C07237=1053.526,42.373,-75.968,170.999,31.827,155.969
C07238=1053.520,42.124,-75.951,170.997,31.825,155.968
C07239=1053.514,41.874,-75.935,170.995,31.822,155.968
C07240=1053.507,41.624,-75.918,170.994,31.820,155.968
C07241=1053.501,41.376,-75.902,170.993,31.818,155.967
C07242=1053.495,41.126,-75.885,170.991,31.816,155.967
C07243=1053.489,40.877,-75.869,170.989,31.814,155.967
C07244=1053.482,40.628,-75.852,170.988,31.811,155.966
C07245=1053.476,40.378,-75.835,170.986,31.809,155.966
C07246=1053.470,40.129,-75.819,170.984,31.807,155.966
C07247=1053.464,39.880,-75.803,170.983,31.805,155.965
C07248=1053.459,39.630,-75.787,170.981,31.802,155.965
C07249=1053.452,39.381,-75.769,170.979,31.800,155.965
C07250=1053.446,39.131,-75.753,170.978,31.798,155.964
C07251=1053.440,38.882,-75.736,170.977,31.796,155.964
C07252=1053.435,38.632,-75.720,170.975,31.794,155.964
C07253=1053.428,38.382,-75.703,170.974,31.792,155.963
C07254=1053.422,38.134,-75.686,170.972,31.790,155.963
C07255=1053.416,37.884,-75.670,170.970,31.787,155.963
C07256=1053.410,37.635,-75.654,170.969,31.785,155.962
C07257=1053.403,37.386,-75.638,170.967,31.783,155.962
C07258=1053.397,37.136,-75.622,170.965,31.781,155.962
C07259=1053.391,36.886,-75.605,170.963,31.779,155.961
C07260=1053.385,36.637,-75.589,170.962,31.777,155.961
C07261=1053.378,36.388,-75.572,170.961,31.775,155.961
C07262=1053.372,36.139,-75.556,170.959,31.772,155.960
C07263=1053.366,35.889,-75.539,170.958,31.770,155.960
C07264=1053.359,35.640,-75.524,170.956,31.768,155.960
C07265=1053.353,35.391,-75.507,170.954,31.766,155.960
C07266=1053.347,35.141,-75.491,170.953,31.764,155.959
C07267=1053.341,34.892,-75.475,170.951,31.762,155.959
C07268=1053.335,34.642,-75.458,170.949,31.759,155.958
C07269=1053.328,34.393,-75.442,170.947,31.757,155.958
C07270=1053.322,34.143,-75.426,170.946,31.755,155.958
C07271=1053.316,33.894,-75.410,170.945,31.753,155.958
C07272=1053.310,33.645,-75.394,170.943,31.751,155.957
C07273=1053.304,33.395,-75.377,170.942,31.749,155.957
C07274=1053.298,33.145,-75.361,170.940,31.746,155.957
C07275=1053.291,32.896,-75.345,170.938,31.744,155.956
C07276=1053.285,32.647,-75.329,170.937,31.742,155.956
C07277=1053.279,32.398,-75.313,170.935,31.740,155.956
C07278=1053.273,32.148,-75.296,170.933,31.738,155.955
C07279=1053.267,31.899,-75.280,170.931,31.736,155.955
C07280=1053.261,31.650,-75.264,170.930,31.733,155.955
C07281=1053.254,31.400,-75.248,170.929,31.731,155.954
C07282=1053.248,31.151,-75.232,170.927,31.729,155.954
C07283=1053.242,30.901,-75.215,170.926,31.727,155.954
C07284=1053.236,30.652,-75.199,170.924,31.725,155.953
C07285=1053.230,30.403,-75.183,170.922,31.723,155.953
C07286=1053.224,30.153,-75.167,170.920,31.720,155.953
C07287=1053.217,29.868,-75.149,170.919,31.718,155.952
C07288=1053.209,29.582,-75.130,170.917,31.716,155.952
C07289=1053.203,29.296,-75.112,170.915,31.714,155.952
C07290=1053.196,29.011,-75.094,170.914,31.711,155.951
C07291=1053.189,28.761,-75.077,170.912,31.709,155.951
C07292=1053.184,28.511,-75.062,170.910,31.707,155.951
C07293=1053.177,28.262,-75.046,170.909,31.704,155.950
C07294=1053.171,28.012,-75.030,170.907,31.702,155.950
C07295=1053.165,27.763,-75.013,170.905,31.700,155.950
C07296=1053.158,27.514,-74.998,170.903,31.698,155.949
C07297=1053.153,27.264,-74.982,170.902,31.696,155.949
C07298=1053.146,27.015,-74.966,170.900,31.694,155.949
C07299=1053.140,26.765,-74.950,170.899,31.692,155.949
C07300=1053.134,26.516,-74.934,170.897,31.690,155.948
C07301=1053.127,26.267,-74.918,170.896,31.688,155.948
C07302=1053.122,26.017,-74.903,170.894,31.686,155.948
C07303=1053.114,25.767,-74.887,170.892,31.684,155.947
C07304=1053.108,25.518,-74.870,170.891,31.682,155.947
C07305=1053.103,25.269,-74.854,170.889,31.679,155.947
C07306=1053.096,25.019,-74.839,170.887,31.677,155.946
C07307=1053.090,24.770,-74.823,170.885,31.675,155.946
C07308=1053.084,24.521,-74.807,170.884,31.673,155.946
C07309=1053.078,24.271,-74.792,170.883,31.671,155.945
C07310=1053.071,24.022,-74.776,170.881,31.669,155.945
C07311=1053.065,23.772,-74.760,170.880,31.667,155.945
C07312=1053.059,23.523,-74.744,170.878,31.665,155.945
C07313=1053.053,23.273,-74.729,170.876,31.663,155.944
C07314=1053.047,23.024,-74.712,170.874,31.660,155.944
C07315=1053.040,22.775,-74.697,170.873,31.659,155.944
C07316=1053.035,22.525,-74.681,170.871,31.656,155.943
C07317=1053.028,22.276,-74.666,170.869,31.654,155.943
C07318=1053.022,22.026,-74.650,170.868,31.652,155.943
C07319=1053.016,21.777,-74.634,170.867,31.650,155.942
C07320=1053.010,21.528,-74.618,170.865,31.648,155.942
C07321=1053.003,21.278,-74.603,170.863,31.645,155.942
C07322=1052.997,21.029,-74.587,170.862,31.644,155.942
C07323=1052.991,20.779,-74.571,170.860,31.641,155.941
C07324=1052.985,20.530,-74.556,170.858,31.639,155.941
C07325=1052.979,20.280,-74.539,170.856,31.637,155.941
C07326=1052.973,20.030,-74.525,170.855,31.635,155.940
C07327=1052.967,19.781,-74.508,170.853,31.633,155.940
C07328=1052.960,19.531,-74.493,170.852,31.631,155.940
C07329=1052.954,19.282,-74.478,170.850,31.629,155.939
C07330=1052.948,19.032,-74.462,170.849,31.627,155.939
C07331=1052.941,18.783,-74.446,170.847,31.625,155.939
C07332=1052.936,18.533,-74.431,170.845,31.623,155.939
C07333=1052.929,18.284,-74.415,170.843,31.621,155.938
C07334=1052.923,18.035,-74.400,170.842,31.619,155.938
C07335=1052.917,17.785,-74.384,170.840,31.617,155.938
C07336=1052.910,17.536,-74.369,170.838,31.615,155.937
C07337=1052.905,17.287,-74.353,170.837,31.613,155.937
C07338=1052.898,17.037,-74.338,170.836,31.611,155.937
C07339=1052.892,16.788,-74.323,170.834,31.608,155.936
C07340=1052.886,16.538,-74.307,170.832,31.606,155.936
C07341=1052.879,16.289,-74.291,170.830,31.604,155.936
C07342=1052.874,16.039,-74.276,170.829,31.602,155.936
C07343=1052.867,15.790,-74.260,170.827,31.600,155.935
C07344=1052.861,15.541,-74.245,170.825,31.598,155.935
C07345=1052.855,15.291,-74.230,170.823,31.596,155.935
C07346=1052.848,15.042,-74.214,170.823,31.594,155.934
C07347=1052.842,14.792,-74.199,170.821,31.592,155.934
C07348=1052.836,14.543,-74.183,170.819,31.590,155.934
C07349=1052.830,14.294,-74.168,170.817,31.588,155.934
C07350=1052.824,14.044,-74.153,170.816,31.586,155.933
C07351=1052.816,13.760,-74.135,170.814,31.584,155.933
C07352=1052.809,13.475,-74.118,170.812,31.581,155.933
C07353=1052.802,13.191,-74.100,170.810,31.579,155.932
C07354=1052.795,12.906,-74.083,170.808,31.577,155.932
C07355=1052.789,12.656,-74.068,170.807,31.575,155.932
C07356=1052.782,12.407,-74.052,170.805,31.573,155.931
C07357=1052.776,12.158,-74.037,170.803,31.571,155.931
C07358=1052.769,11.908,-74.022,170.802,31.569,155.931
C07359=1052.764,11.658,-74.007,170.800,31.566,155.931
C07360=1052.757,11.409,-73.991,170.798,31.564,155.930
C07361=1052.751,11.160,-73.977,170.796,31.563,155.930
C07362=1052.745,10.910,-73.962,170.794,31.561,155.930
C07363=1052.738,10.661,-73.946,170.793,31.559,155.929
C07364=1052.732,10.412,-73.931,170.792,31.557,155.929
C07365=1052.725,10.162,-73.916,170.790,31.555,155.929
C07366=1052.719,9.912,-73.901,170.788,31.553,155.929
C07367=1052.713,9.662,-73.886,170.787,31.551,155.928
C07368=1052.707,9.414,-73.870,170.785,31.548,155.928
C07369=1052.701,9.164,-73.855,170.783,31.547,155.928
C07370=1052.695,8.915,-73.841,170.781,31.545,155.928
C07371=1052.688,8.665,-73.826,170.779,31.543,155.927
C07372=1052.682,8.415,-73.811,170.778,31.541,155.927
C07373=1052.675,8.166,-73.795,170.777,31.539,155.927
C07374=1052.669,7.917,-73.780,170.775,31.537,155.926
C07375=1052.664,7.668,-73.765,170.773,31.534,155.926
C07376=1052.657,7.418,-73.750,170.772,31.533,155.926
C07377=1052.651,7.168,-73.735,170.770,31.531,155.926
C07378=1052.645,6.919,-73.720,170.768,31.529,155.925
C07379=1052.638,6.669,-73.705,170.766,31.527,155.925
C07380=1052.632,6.421,-73.690,170.764,31.525,155.925
C07381=1052.626,6.171,-73.675,170.763,31.523,155.924
C07382=1052.619,5.921,-73.660,170.762,31.521,155.924
C07383=1052.613,5.672,-73.645,170.760,31.519,155.924
C07384=1052.607,5.422,-73.630,170.758,31.516,155.924
C07385=1052.602,5.173,-73.615,170.757,31.515,155.923
C07386=1052.595,4.923,-73.600,170.755,31.513,155.923
C07387=1052.589,4.673,-73.585,170.753,31.511,155.923
C07388=1052.582,4.424,-73.570,170.751,31.509,155.922
C07389=1052.577,4.175,-73.555,170.749,31.507,155.922
C07390=1052.570,3.925,-73.540,170.749,31.505,155.922
C07391=1052.564,3.675,-73.525,170.747,31.503,155.922
C07392=1052.557,3.426,-73.511,170.745,31.500,155.921
C07393=1052.552,3.177,-73.496,170.743,31.499,155.921
C07394=1052.545,2.927,-73.481,170.741,31.497,155.921
C07395=1052.539,2.678,-73.466,170.740,31.495,155.921
C07396=1052.533,2.429,-73.451,170.738,31.493,155.920
C07397=1052.527,2.179,-73.437,170.736,31.491,155.920
C07398=1052.521,1.929,-73.421,170.734,31.489,155.920
C07399=1052.515,1.679,-73.406,170.733,31.487,155.919
C07400=1052.509,1.430,-73.391,170.732,31.485,155.919
C07401=1052.503,1.181,-73.377,170.730,31.483,155.919
C07402=1052.496,0.931,-73.362,170.728,31.481,155.919
C07403=1052.490,0.682,-73.347,170.726,31.479,155.918
C07404=1052.484,0.432,-73.332,170.725,31.477,155.918
C07405=1052.478,0.183,-73.317,170.723,31.475,155.918
C07406=1052.472,-0.066,-73.303,170.721,31.473,155.917
C07407=1052.465,-0.316,-73.288,170.719,31.471,155.917
C07408=1052.459,-0.566,-73.273,170.718,31.469,155.917
C07409=1052.453,-0.814,-73.258,170.717,31.467,155.917
C07410=1052.447,-1.065,-73.244,170.715,31.465,155.916
C07411=1052.441,-1.314,-73.229,170.713,31.463,155.916
C07412=1052.435,-1.563,-73.214,170.711,31.461,155.916
C07413=1052.429,-1.813,-73.199,170.709,31.459,155.916
C07414=1052.422,-2.063,-73.184,170.708,31.457,155.915
C07415=1052.415,-2.345,-73.168,170.705,31.454,155.915
C07416=1052.409,-2.628,-73.152,170.704,31.452,155.915
C07417=1052.402,-2.910,-73.135,170.702,31.450,155.914
C07418=1052.395,-3.193,-73.118,170.700,31.447,155.914
C07419=1052.389,-3.442,-73.103,170.699,31.446,155.914
C07420=1052.383,-3.692,-73.089,170.697,31.444,155.914
C07421=1052.377,-3.941,-73.074,170.695,31.442,155.913
C07422=1052.369,-4.191,-73.060,170.693,31.440,155.913
C07423=1052.364,-4.440,-73.045,170.691,31.438,155.913
C07424=1052.358,-4.690,-73.031,170.690,31.436,155.912
C07425=1052.351,-4.940,-73.016,170.689,31.435,155.912
C07426=1052.345,-5.188,-73.002,170.687,31.433,155.912
C07427=1052.338,-5.438,-72.987,170.685,31.431,155.912
C07428=1052.333,-5.688,-72.973,170.683,31.429,155.912
C07429=1052.326,-5.937,-72.958,170.681,31.427,155.911
C07430=1052.319,-6.187,-72.944,170.679,31.425,155.911
C07431=1052.314,-6.436,-72.930,170.678,31.423,155.911
C07432=1052.307,-6.686,-72.915,170.676,31.421,155.911
C07433=1052.301,-6.935,-72.900,170.675,31.419,155.910
C07434=1052.295,-7.185,-72.887,170.673,31.417,155.910
C07435=1052.288,-7.434,-72.872,170.671,31.416,155.910
C07436=1052.283,-7.683,-72.857,170.669,31.414,155.909
C07437=1052.276,-7.933,-72.844,170.667,31.411,155.909
C07438=1052.270,-8.183,-72.829,170.666,31.410,155.909
C07439=1052.264,-8.432,-72.814,170.664,31.408,155.909
C07440=1052.258,-8.682,-72.800,170.662,31.406,155.908
C07441=1052.251,-8.931,-72.786,170.660,31.404,155.908
C07442=1052.245,-9.181,-72.772,170.659,31.402,155.908
C07443=1052.239,-9.431,-72.757,170.657,31.400,155.908
C07444=1052.232,-9.679,-72.743,170.656,31.399,155.907
C07445=1052.226,-9.930,-72.729,170.654,31.397,155.907
C07446=1052.220,-10.179,-72.714,170.652,31.395,155.907
C07447=1052.213,-10.429,-72.700,170.650,31.393,155.907
C07448=1052.208,-10.678,-72.686,170.648,31.391,155.906
C07449=1052.202,-10.928,-72.672,170.646,31.389,155.906
C07450=1052.195,-11.176,-72.658,170.645,31.387,155.906
C07451=1052.189,-11.427,-72.643,170.644,31.385,155.906
C07452=1052.183,-11.676,-72.629,170.642,31.384,155.906
C07453=1052.177,-11.926,-72.615,170.640,31.382,155.905
C07454=1052.171,-12.175,-72.601,170.638,31.380,155.905
C07455=1052.165,-12.425,-72.586,170.636,31.378,155.905
C07456=1052.159,-12.674,-72.572,170.634,31.376,155.905
C07457=1052.152,-12.924,-72.558,170.633,31.374,155.904
C07458=1052.146,-13.173,-72.544,170.631,31.372,155.904
C07459=1052.140,-13.423,-72.529,170.630,31.370,155.904
C07460=1052.134,-13.672,-72.515,170.628,31.368,155.903
C07461=1052.127,-13.922,-72.501,170.626,31.367,155.903
C07462=1052.122,-14.171,-72.487,170.624,31.365,155.903
C07463=1052.115,-14.421,-72.473,170.622,31.362,155.903
C07464=1052.109,-14.670,-72.458,170.621,31.361,155.903
C07465=1052.102,-14.920,-72.445,170.619,31.359,155.902
C07466=1052.097,-15.169,-72.431,170.617,31.358,155.902
C07467=1052.090,-15.419,-72.416,170.616,31.355,155.902
C07468=1052.084,-15.668,-72.403,170.614,31.354,155.902
C07469=1052.077,-15.918,-72.388,170.612,31.352,155.901
C07470=1052.072,-16.167,-72.374,170.610,31.350,155.901
C07471=1052.065,-16.417,-72.361,170.608,31.348,155.901
C07472=1052.059,-16.666,-72.346,170.606,31.347,155.901
C07473=1052.052,-16.916,-72.333,170.605,31.345,155.900
C07474=1052.047,-17.166,-72.319,170.603,31.343,155.900
C07475=1052.040,-17.415,-72.304,170.602,31.341,155.900
C07476=1052.034,-17.665,-72.291,170.600,31.340,155.900
C07477=1052.027,-17.915,-72.277,170.598,31.337,155.900
C07478=1052.021,-18.164,-72.264,170.596,31.336,155.899
C07479=1052.014,-18.445,-72.248,170.594,31.334,155.899
C07480=1052.007,-18.725,-72.231,170.592,31.332,155.899
C07481=1052.000,-19.007,-72.216,170.590,31.330,155.898
C07482=1051.993,-19.288,-72.200,170.588,31.327,155.898
C07483=1051.987,-19.537,-72.187,170.586,31.326,155.898
C07484=1051.980,-19.787,-72.173,170.585,31.324,155.898
C07485=1051.975,-20.036,-72.159,170.583,31.322,155.898
C07486=1051.967,-20.286,-72.145,170.581,31.320,155.897
C07487=1051.962,-20.535,-72.131,170.579,31.319,155.897
C07488=1051.956,-20.785,-72.118,170.577,31.317,155.897
C07489=1051.949,-21.035,-72.104,170.575,31.315,155.897
C07490=1051.943,-21.284,-72.090,170.574,31.314,155.896
C07491=1051.936,-21.534,-72.076,170.572,31.312,155.896
C07492=1051.931,-21.783,-72.062,170.571,31.310,155.896
C07493=1051.925,-22.032,-72.049,170.569,31.308,155.896
C07494=1051.918,-22.282,-72.035,170.567,31.306,155.896
C07495=1051.912,-22.532,-72.021,170.565,31.304,155.895
C07496=1051.906,-22.781,-72.008,170.563,31.303,155.895
C07497=1051.900,-23.031,-71.993,170.561,31.301,155.895
C07498=1051.894,-23.280,-71.980,170.559,31.299,155.895
C07499=1051.887,-23.529,-71.966,170.557,31.297,155.894
C07500=1051.881,-23.780,-71.952,170.557,31.296,155.894
C07501=1051.875,-24.029,-71.939,170.555,31.293,155.894
C07502=1051.869,-24.278,-71.926,170.553,31.292,155.894
C07503=1051.863,-24.528,-71.911,170.551,31.290,155.894
C07504=1051.857,-24.778,-71.898,170.549,31.288,155.893
C07505=1051.850,-25.027,-71.885,170.547,31.287,155.893
C07506=1051.844,-25.277,-71.871,170.545,31.285,155.893
C07507=1051.838,-25.526,-71.857,170.543,31.283,155.893
C07508=1051.832,-25.775,-71.843,170.542,31.281,155.892
C07509=1051.825,-26.025,-71.829,170.540,31.280,155.892
C07510=1051.819,-26.275,-71.816,170.538,31.277,155.892
C07511=1051.814,-26.524,-71.802,170.537,31.276,155.892
C07512=1051.807,-26.774,-71.788,170.535,31.275,155.892
C07513=1051.801,-27.024,-71.775,170.533,31.272,155.891
C07514=1051.795,-27.273,-71.762,170.531,31.271,155.891
C07515=1051.788,-27.523,-71.748,170.529,31.269,155.891
C07516=1051.782,-27.772,-71.734,170.527,31.267,155.891
C07517=1051.776,-28.022,-71.721,170.526,31.266,155.891
C07518=1051.769,-28.272,-71.707,170.524,31.264,155.890
C07519=1051.763,-28.521,-71.695,170.522,31.262,155.890
C07520=1051.757,-28.771,-71.682,170.520,31.261,155.890
C07521=1051.751,-29.020,-71.668,170.518,31.259,155.890
C07522=1051.744,-29.270,-71.655,170.516,31.258,155.890
C07523=1051.739,-29.520,-71.641,170.514,31.255,155.889
C07524=1051.732,-29.769,-71.628,170.512,31.254,155.889
C07525=1051.726,-30.019,-71.614,170.511,31.252,155.889
C07526=1051.719,-30.268,-71.601,170.510,31.250,155.889
C07527=1051.713,-30.517,-71.587,170.508,31.249,155.888
C07528=1051.707,-30.767,-71.574,170.506,31.247,155.888
C07529=1051.700,-31.017,-71.561,170.504,31.246,155.888
C07530=1051.694,-31.266,-71.548,170.502,31.244,155.888
C07531=1051.688,-31.516,-71.535,170.500,31.242,155.888
C07532=1051.682,-31.765,-71.521,170.498,31.241,155.888
C07533=1051.676,-32.015,-71.507,170.496,31.239,155.887
C07534=1051.669,-32.264,-71.494,170.495,31.237,155.887
C07535=1051.664,-32.514,-71.481,170.493,31.236,155.887
C07536=1051.657,-32.764,-71.468,170.491,31.234,155.887
C07537=1051.651,-33.014,-71.454,170.489,31.232,155.887
C07538=1051.644,-33.263,-71.441,170.487,31.230,155.886
C07539=1051.638,-33.512,-71.428,170.485,31.229,155.886
C07540=1051.632,-33.762,-71.415,170.483,31.227,155.886
C07541=1051.626,-34.011,-71.402,170.481,31.226,155.886
C07542=1051.619,-34.261,-71.388,170.480,31.224,155.886
C07543=1051.613,-34.542,-71.373,170.478,31.222,155.885
C07544=1051.606,-34.822,-71.358,170.476,31.220,155.885
C07545=1051.599,-35.102,-71.344,170.474,31.218,155.885
C07546=1051.592,-35.382,-71.329,170.472,31.216,155.885
C07547=1051.586,-35.632,-71.316,170.470,31.215,155.884
C07548=1051.580,-35.881,-71.303,170.468,31.213,155.884
C07549=1051.573,-36.130,-71.290,170.466,31.212,155.884
C07550=1051.567,-36.380,-71.277,170.465,31.210,155.884
C07551=1051.561,-36.630,-71.263,170.463,31.208,155.884
C07552=1051.554,-36.879,-71.250,170.461,31.207,155.884
C07553=1051.548,-37.129,-71.238,170.459,31.205,155.883
C07554=1051.542,-37.379,-71.224,170.457,31.203,155.883
C07555=1051.537,-37.628,-71.211,170.455,31.201,155.883
C07556=1051.531,-37.878,-71.198,170.453,31.200,155.883
C07557=1051.525,-38.127,-71.185,170.451,31.198,155.883
C07558=1051.518,-38.376,-71.171,170.449,31.197,155.882
C07559=1051.512,-38.627,-71.159,170.448,31.195,155.882
C07560=1051.506,-38.876,-71.145,170.446,31.193,155.882
C07561=1051.499,-39.126,-71.133,170.444,31.192,155.882
C07562=1051.493,-39.375,-71.120,170.442,31.190,155.882
C07563=1051.487,-39.624,-71.107,170.440,31.189,155.881
C07564=1051.481,-39.874,-71.094,170.438,31.187,155.881
C07565=1051.475,-40.124,-71.081,170.436,31.186,155.881
C07566=1051.468,-40.374,-71.068,170.434,31.184,155.881
C07567=1051.461,-40.623,-71.055,170.433,31.183,155.881
C07568=1051.455,-40.873,-71.043,170.431,31.181,155.881
C07569=1051.449,-41.122,-71.030,170.429,31.180,155.880
C07570=1051.443,-41.372,-71.017,170.427,31.178,155.880
C07571=1051.437,-41.621,-71.004,170.425,31.177,155.880
C07572=1051.430,-41.871,-70.992,170.423,31.175,155.880
C07573=1051.424,-42.120,-70.978,170.421,31.173,155.880
C07574=1051.418,-42.370,-70.966,170.419,31.171,155.880
C07575=1051.411,-42.620,-70.952,170.417,31.170,155.879
C07576=1051.405,-42.870,-70.940,170.416,31.168,155.879
C07577=1051.399,-43.119,-70.926,170.414,31.167,155.879
C07578=1051.392,-43.369,-70.914,170.412,31.165,155.879
C07579=1051.386,-43.618,-70.901,170.410,31.164,155.879
C07580=1051.380,-43.868,-70.889,170.408,31.162,155.879
C07581=1051.374,-44.118,-70.876,170.406,31.161,155.878
C07582=1051.367,-44.367,-70.863,170.404,31.159,155.878
C07583=1051.362,-44.617,-70.851,170.402,31.158,155.878
C07584=1051.355,-44.866,-70.838,170.401,31.156,155.878
C07585=1051.349,-45.116,-70.825,170.399,31.155,155.878
C07586=1051.344,-45.366,-70.813,170.397,31.153,155.878
C07587=1051.337,-45.615,-70.800,170.395,31.152,155.877
C07588=1051.331,-45.865,-70.787,170.393,31.150,155.877
C07589=1051.324,-46.114,-70.774,170.391,31.148,155.877
C07590=1051.319,-46.364,-70.761,170.389,31.147,155.877
C07591=1051.312,-46.613,-70.749,170.387,31.145,155.877
C07592=1051.306,-46.863,-70.736,170.385,31.144,155.877
C07593=1051.300,-47.112,-70.724,170.384,31.142,155.876
C07594=1051.294,-47.362,-70.711,170.382,31.141,155.876
C07595=1051.288,-47.612,-70.698,170.380,31.139,155.876
C07596=1051.281,-47.861,-70.686,170.378,31.138,155.876
C07597=1051.275,-48.111,-70.673,170.376,31.136,155.876
C07598=1051.269,-48.361,-70.661,170.374,31.135,155.876
C07599=1051.263,-48.610,-70.648,170.372,31.133,155.875
C07600=1051.256,-48.860,-70.636,170.370,31.132,155.875
C07601=1051.250,-49.110,-70.623,170.369,31.130,155.875
C07602=1051.245,-49.360,-70.610,170.367,31.129,155.875
C07603=1051.238,-49.609,-70.597,170.365,31.127,155.875
C07604=1051.232,-49.858,-70.585,170.363,31.126,155.875
C07605=1051.226,-50.108,-70.573,170.361,31.125,155.875
C07606=1051.220,-50.358,-70.560,170.359,31.123,155.874
C07607=1051.212,-50.639,-70.547,170.357,31.122,155.874
C07608=1051.205,-50.919,-70.532,170.354,31.120,155.874
C07609=1051.198,-51.199,-70.518,170.352,31.118,155.874
C07610=1051.191,-51.480,-70.504,170.351,31.117,155.874
C07611=1051.184,-51.729,-70.492,170.349,31.115,155.874
C07612=1051.178,-51.979,-70.480,170.347,31.114,155.873
C07613=1051.172,-52.229,-70.468,170.345,31.112,155.873
C07614=1051.166,-52.479,-70.455,170.343,31.111,155.873
C07615=1051.159,-52.728,-70.443,170.341,31.110,155.873
C07616=1051.153,-52.978,-70.431,170.339,31.108,155.873
C07617=1051.147,-53.228,-70.419,170.337,31.107,155.873
C07618=1051.140,-53.477,-70.406,170.334,31.106,155.873
C07619=1051.134,-53.726,-70.394,170.333,31.104,155.872
C07620=1051.127,-53.976,-70.382,170.331,31.103,155.872
C07621=1051.121,-54.226,-70.369,170.329,31.102,155.872
C07622=1051.115,-54.476,-70.357,170.327,31.100,155.872
C07623=1051.108,-54.725,-70.345,170.325,31.099,155.872
C07624=1051.103,-54.974,-70.333,170.323,31.098,155.872
C07625=1051.096,-55.224,-70.321,170.321,31.096,155.872
C07626=1051.090,-55.474,-70.308,170.319,31.095,155.872
C07627=1051.083,-55.723,-70.297,170.317,31.094,155.872
C07628=1051.077,-55.973,-70.285,170.316,31.092,155.871
C07629=1051.071,-56.223,-70.272,170.314,31.091,155.871
C07630=1051.064,-56.472,-70.260,170.312,31.089,155.871
C07631=1051.058,-56.722,-70.247,170.310,31.088,155.871
C07632=1051.052,-56.972,-70.236,170.308,31.087,155.871
C07633=1051.045,-57.221,-70.224,170.306,31.085,155.871
C07634=1051.040,-57.471,-70.211,170.304,31.084,155.871
C07635=1051.033,-57.720,-70.199,170.301,31.083,155.870
C07636=1051.026,-57.970,-70.187,170.300,31.081,155.870
C07637=1051.021,-58.220,-70.175,170.298,31.080,155.870
C07638=1051.014,-58.469,-70.163,170.296,31.079,155.870
C07639=1051.008,-58.719,-70.150,170.294,31.078,155.870
C07640=1051.002,-58.969,-70.139,170.292,31.076,155.870
C07641=1050.996,-59.218,-70.128,170.290,31.075,155.870
C07642=1050.990,-59.468,-70.115,170.288,31.074,155.870
C07643=1050.983,-59.718,-70.103,170.286,31.072,155.869
C07644=1050.976,-59.967,-70.091,170.284,31.071,155.869
C07645=1050.971,-60.217,-70.079,170.282,31.070,155.869
C07646=1050.964,-60.467,-70.067,170.281,31.068,155.869
C07647=1050.958,-60.715,-70.055,170.279,31.067,155.869
C07648=1050.952,-60.966,-70.043,170.277,31.066,155.869
C07649=1050.946,-61.215,-70.031,170.275,31.064,155.869
C07650=1050.939,-61.465,-70.019,170.272,31.063,155.869
C07651=1050.934,-61.714,-70.007,170.270,31.062,155.869
C07652=1050.927,-61.964,-69.995,170.268,31.060,155.868
C07653=1050.920,-62.213,-69.983,170.266,31.059,155.868
C07654=1050.915,-62.464,-69.971,170.264,31.058,155.868
C07655=1050.908,-62.713,-69.959,170.263,31.057,155.868
C07656=1050.902,-62.962,-69.948,170.261,31.055,155.868
C07657=1050.896,-63.212,-69.935,170.259,31.054,155.868
C07658=1050.890,-63.462,-69.924,170.257,31.053,155.868
C07659=1050.883,-63.712,-69.912,170.255,31.051,155.868
C07660=1050.878,-63.961,-69.900,170.253,31.050,155.868
C07661=1050.871,-64.211,-69.888,170.251,31.049,155.867
C07662=1050.865,-64.461,-69.877,170.248,31.048,155.867
C07663=1050.860,-64.710,-69.864,170.246,31.046,155.867
C07664=1050.853,-64.960,-69.852,170.245,31.045,155.867
C07665=1050.846,-65.209,-69.840,170.243,31.044,155.867
C07666=1050.840,-65.459,-69.829,170.241,31.042,155.867
C07667=1050.835,-65.709,-69.817,170.239,31.041,155.867
C07668=1050.828,-65.958,-69.805,170.237,31.040,155.867
C07669=1050.822,-66.208,-69.794,170.235,31.039,155.867
C07670=1050.816,-66.458,-69.782,170.233,31.037,155.866
C07671=1050.809,-66.739,-69.769,170.230,31.036,155.866
C07672=1050.801,-67.021,-69.755,170.228,31.035,155.866
C07673=1050.795,-67.303,-69.742,170.227,31.033,155.866
C07674=1050.788,-67.585,-69.728,170.224,31.032,155.866
C07675=1050.782,-67.835,-69.717,170.222,31.031,155.866
C07676=1050.776,-68.084,-69.706,170.220,31.029,155.866
C07677=1050.770,-68.334,-69.693,170.218,31.028,155.866
C07678=1050.764,-68.585,-69.682,170.216,31.027,155.865
C07679=1050.758,-68.833,-69.670,170.214,31.026,155.865
C07680=1050.751,-69.083,-69.658,170.212,31.024,155.865
C07681=1050.745,-69.333,-69.646,170.210,31.023,155.865
C07682=1050.739,-69.582,-69.635,170.209,31.022,155.865
C07683=1050.733,-69.833,-69.624,170.207,31.021,155.865
C07684=1050.727,-70.081,-69.612,170.204,31.019,155.865
C07685=1050.721,-70.332,-69.600,170.202,31.018,155.865
C07686=1050.715,-70.581,-69.588,170.200,31.017,155.865
C07687=1050.709,-70.831,-69.577,170.198,31.016,155.865
C07688=1050.702,-71.081,-69.565,170.196,31.014,155.864
C07689=1050.697,-71.330,-69.553,170.194,31.013,155.864
C07690=1050.691,-71.580,-69.542,170.192,31.012,155.864
C07691=1050.685,-71.829,-69.530,170.191,31.011,155.864
C07692=1050.678,-72.079,-69.519,170.189,31.009,155.864
C07693=1050.673,-72.329,-69.507,170.187,31.008,155.864
C07694=1050.667,-72.578,-69.496,170.184,31.007,155.864
C07695=1050.660,-72.829,-69.484,170.182,31.006,155.864
C07696=1050.654,-73.077,-69.473,170.180,31.005,155.864
C07697=1050.648,-73.328,-69.462,170.178,31.003,155.864
C07698=1050.643,-73.577,-69.449,170.176,31.002,155.864
C07699=1050.636,-73.827,-69.438,170.174,31.001,155.863
C07700=1050.630,-74.076,-69.427,170.173,31.000,155.863
C07701=1050.624,-74.326,-69.415,170.171,30.999,155.863
C07702=1050.618,-74.576,-69.404,170.169,30.998,155.863
C07703=1050.611,-74.825,-69.393,170.166,30.996,155.863
C07704=1050.605,-75.075,-69.381,170.164,30.995,155.863
C07705=1050.599,-75.325,-69.370,170.162,30.995,155.863
C07706=1050.593,-75.574,-69.358,170.160,30.994,155.863
C07707=1050.587,-75.824,-69.348,170.158,30.992,155.863
C07708=1050.580,-76.073,-69.336,170.156,30.991,155.863
C07709=1050.574,-76.324,-69.324,170.154,30.990,155.863
C07710=1050.568,-76.573,-69.313,170.152,30.989,155.863
C07711=1050.562,-76.823,-69.302,170.150,30.988,155.862
C07712=1050.556,-77.072,-69.291,170.148,30.987,155.862
C07713=1050.550,-77.322,-69.279,170.146,30.986,155.862
C07714=1050.544,-77.572,-69.269,170.144,30.985,155.862
C07715=1050.537,-77.821,-69.257,170.142,30.983,155.862
C07716=1050.531,-78.071,-69.246,170.140,30.982,155.862
C07717=1050.525,-78.321,-69.234,170.138,30.981,155.862
C07718=1050.519,-78.571,-69.224,170.135,30.980,155.862
C07719=1050.513,-78.820,-69.212,170.133,30.979,155.862
C07720=1050.506,-79.069,-69.201,170.132,30.978,155.862
C07721=1050.500,-79.319,-69.190,170.130,30.977,155.862
C07722=1050.494,-79.569,-69.179,170.128,30.976,155.862
C07723=1050.487,-79.819,-69.167,170.126,30.975,155.862
C07724=1050.482,-80.068,-69.156,170.124,30.974,155.862
C07725=1050.475,-80.318,-69.145,170.121,30.973,155.862
C07726=1050.470,-80.568,-69.134,170.119,30.972,155.862
C07727=1050.463,-80.818,-69.124,170.117,30.971,155.862
C07728=1050.457,-81.067,-69.113,170.115,30.970,155.861
C07729=1050.450,-81.317,-69.101,170.113,30.969,155.861
C07730=1050.444,-81.566,-69.090,170.112,30.969,155.861
C07731=1050.437,-81.816,-69.079,170.109,30.967,155.861
C07732=1050.432,-82.066,-69.068,170.107,30.967,155.861
C07733=1050.425,-82.316,-69.057,170.105,30.966,155.861
C07734=1050.419,-82.565,-69.047,170.103,30.965,155.861
C07735=1050.412,-82.849,-69.034,170.100,30.964,155.861
C07736=1050.405,-83.133,-69.022,170.098,30.963,155.861
C07737=1050.398,-83.417,-69.009,170.096,30.961,155.861
C07738=1050.391,-83.702,-68.997,170.093,30.960,155.861
C07739=1050.384,-83.951,-68.986,170.091,30.959,155.861
C07740=1050.378,-84.200,-68.975,170.090,30.958,155.861
C07741=1050.372,-84.451,-68.963,170.088,30.957,155.861
C07742=1050.366,-84.700,-68.953,170.085,30.956,155.861
C07743=1050.359,-84.950,-68.942,170.083,30.955,155.861
C07744=1050.353,-85.199,-68.931,170.081,30.955,155.861
C07745=1050.347,-85.449,-68.920,170.079,30.954,155.861
C07746=1050.340,-85.699,-68.910,170.077,30.953,155.861
C07747=1050.334,-85.948,-68.899,170.075,30.952,155.861
C07748=1050.328,-86.198,-68.887,170.072,30.951,155.861
C07749=1050.322,-86.448,-68.877,170.070,30.950,155.861
C07750=1050.316,-86.697,-68.866,170.069,30.949,155.861
C07751=1050.310,-86.947,-68.855,170.067,30.948,155.860
C07752=1050.303,-87.197,-68.845,170.065,30.947,155.860
C07753=1050.297,-87.447,-68.834,170.063,30.947,155.860
C07754=1050.291,-87.697,-68.823,170.060,30.945,155.860
C07755=1050.285,-87.946,-68.813,170.058,30.945,155.860
C07756=1050.278,-88.196,-68.802,170.056,30.944,155.860
C07757=1050.273,-88.446,-68.791,170.054,30.943,155.860
C07758=1050.266,-88.695,-68.781,170.052,30.942,155.860
C07759=1050.260,-88.945,-68.769,170.050,30.941,155.860
C07760=1050.254,-89.194,-68.759,170.047,30.940,155.860
C07761=1050.248,-89.444,-68.748,170.046,30.939,155.860
C07762=1050.241,-89.694,-68.737,170.044,30.939,155.860
C07763=1050.236,-89.944,-68.727,170.042,30.938,155.860
C07764=1050.229,-90.193,-68.717,170.040,30.937,155.860
C07765=1050.223,-90.443,-68.705,170.037,30.936,155.860
C07766=1050.217,-90.693,-68.694,170.035,30.935,155.860
C07767=1050.211,-90.942,-68.684,170.033,30.934,155.860
C07768=1050.205,-91.192,-68.673,170.031,30.933,155.860
C07769=1050.198,-91.442,-68.663,170.029,30.933,155.860
C07770=1050.193,-91.691,-68.652,170.027,30.932,155.860
C07771=1050.187,-91.941,-68.642,170.024,30.931,155.860
C07772=1050.180,-92.191,-68.631,170.023,30.930,155.860
C07773=1050.174,-92.440,-68.620,170.021,30.929,155.860
C07774=1050.169,-92.690,-68.610,170.019,30.928,155.860
C07775=1050.162,-92.940,-68.600,170.017,30.927,155.860
C07776=1050.156,-93.190,-68.588,170.014,30.927,155.860
C07777=1050.149,-93.439,-68.578,170.012,30.926,155.860
C07778=1050.144,-93.689,-68.568,170.010,30.925,155.860
C07779=1050.138,-93.939,-68.557,170.008,30.924,155.860
C07780=1050.131,-94.188,-68.546,170.006,30.923,155.860
C07781=1050.125,-94.438,-68.536,170.004,30.923,155.860
C07782=1050.119,-94.688,-68.526,170.001,30.922,155.860
C07783=1050.113,-94.937,-68.515,170.000,30.921,155.860
C07784=1050.107,-95.187,-68.504,169.998,30.920,155.860
C07785=1050.101,-95.437,-68.494,169.996,30.920,155.860
C07786=1050.095,-95.687,-68.483,169.994,30.919,155.860
C07787=1050.089,-95.936,-68.473,169.991,30.918,155.860
C07788=1050.083,-96.186,-68.463,169.989,30.917,155.860
C07789=1050.077,-96.436,-68.452,169.987,30.917,155.860
C07790=1050.070,-96.685,-68.441,169.985,30.916,155.860
C07791=1050.065,-96.936,-68.431,169.983,30.915,155.860
C07792=1050.059,-97.185,-68.421,169.981,30.914,155.860
C07793=1050.053,-97.434,-68.410,169.978,30.913,155.860
C07794=1050.047,-97.684,-68.401,169.977,30.912,155.860
C07795=1050.040,-97.934,-68.389,169.975,30.911,155.860
C07796=1050.034,-98.184,-68.380,169.973,30.911,155.860
C07797=1050.028,-98.433,-68.369,169.970,30.910,155.860
C07798=1050.022,-98.683,-68.359,169.968,30.910,155.860
C07799=1050.015,-98.970,-68.347,169.966,30.909,155.860
C07800=1050.008,-99.256,-68.336,169.963,30.908,155.860
C07801=1050.001,-99.542,-68.324,169.961,30.907,155.860
C07802=1049.993,-99.829,-68.312,169.958,30.906,155.860
C07803=1049.987,-100.078,-68.301,169.956,30.906,155.860
C07804=1049.981,-100.328,-68.292,169.954,30.905,155.860
C07805=1049.975,-100.577,-68.281,169.952,30.905,155.860
C07806=1049.969,-100.828,-68.271,169.950,30.904,155.860
C07807=1049.962,-101.077,-68.261,169.948,30.903,155.860
C07808=1049.956,-101.327,-68.251,169.946,30.902,155.860
C07809=1049.950,-101.577,-68.241,169.944,30.902,155.860
C07810=1049.944,-101.826,-68.231,169.941,30.901,155.860
C07811=1049.938,-102.076,-68.221,169.939,30.901,155.860
C07812=1049.932,-102.325,-68.210,169.937,30.900,155.860
C07813=1049.926,-102.575,-68.201,169.935,30.900,155.860
C07814=1049.919,-102.825,-68.190,169.933,30.899,155.860
C07815=1049.913,-103.075,-68.180,169.930,30.898,155.860
C07816=1049.907,-103.324,-68.170,169.928,30.897,155.860
C07817=1049.901,-103.574,-68.160,169.926,30.897,155.860
C07818=1049.895,-103.824,-68.150,169.925,30.896,155.860
C07819=1049.889,-104.073,-68.140,169.922,30.896,155.860
C07820=1049.883,-104.323,-68.130,169.920,30.895,155.860
C07821=1049.876,-104.573,-68.120,169.918,30.894,155.860
C07822=1049.871,-104.823,-68.110,169.916,30.894,155.860
C07823=1049.865,-105.072,-68.100,169.914,30.893,155.860
C07824=1049.857,-105.322,-68.089,169.911,30.893,155.860
C07825=1049.851,-105.572,-68.080,169.909,30.892,155.860
C07826=1049.846,-105.822,-68.070,169.907,30.891,155.860
C07827=1049.840,-106.072,-68.060,169.905,30.891,155.860
C07828=1049.833,-106.321,-68.050,169.903,30.890,155.860
C07829=1049.827,-106.571,-68.040,169.900,30.890,155.860
C07830=1049.822,-106.821,-68.030,169.898,30.889,155.860
C07831=1049.815,-107.070,-68.020,169.897,30.888,155.860
C07832=1049.809,-107.320,-68.010,169.895,30.888,155.860
C07833=1049.803,-107.570,-68.001,169.892,30.888,155.860
C07834=1049.797,-107.820,-67.991,169.890,30.887,155.860
C07835=1049.791,-108.069,-67.980,169.888,30.886,155.860
C07836=1049.785,-108.319,-67.971,169.886,30.886,155.860
C07837=1049.779,-108.569,-67.961,169.883,30.885,155.860
C07838=1049.772,-108.818,-67.951,169.881,30.885,155.860
C07839=1049.766,-109.068,-67.941,169.879,30.884,155.861
C07840=1049.760,-109.317,-67.932,169.877,30.884,155.861
C07841=1049.754,-109.567,-67.922,169.875,30.884,155.861
C07842=1049.747,-109.817,-67.912,169.872,30.883,155.861
C07843=1049.742,-110.067,-67.902,169.870,30.882,155.861
C07844=1049.736,-110.317,-67.893,169.869,30.882,155.861
C07845=1049.729,-110.566,-67.882,169.867,30.882,155.861
C07846=1049.723,-110.816,-67.873,169.864,30.881,155.861
C07847=1049.717,-111.066,-67.863,169.862,30.880,155.861
C07848=1049.711,-111.316,-67.854,169.860,30.880,155.861
C07849=1049.705,-111.565,-67.844,169.858,30.880,155.861
C07850=1049.698,-111.815,-67.835,169.855,30.879,155.861
C07851=1049.692,-112.065,-67.825,169.853,30.878,155.861
C07852=1049.686,-112.314,-67.815,169.851,30.878,155.861
C07853=1049.680,-112.564,-67.805,169.849,30.878,155.861
C07854=1049.674,-112.814,-67.795,169.846,30.877,155.861
C07855=1049.668,-113.064,-67.785,169.844,30.877,155.861
C07856=1049.662,-113.314,-67.776,169.842,30.877,155.861
C07857=1049.656,-113.563,-67.766,169.840,30.876,155.861
C07858=1049.649,-113.813,-67.757,169.838,30.875,155.861
C07859=1049.643,-114.063,-67.747,169.836,30.875,155.862
C07860=1049.637,-114.313,-67.738,169.834,30.875,155.862
C07861=1049.631,-114.563,-67.728,169.832,30.874,155.862
C07862=1049.625,-114.812,-67.718,169.829,30.874,155.862
C07863=1049.618,-115.097,-67.708,169.827,30.874,155.862
C07864=1049.611,-115.383,-67.697,169.824,30.873,155.862
C07865=1049.604,-115.668,-67.686,169.822,30.873,155.862
C07866=1049.597,-115.953,-67.675,169.819,30.872,155.862
C07867=1049.591,-116.202,-67.666,169.817,30.872,155.862
C07868=1049.585,-116.452,-67.656,169.815,30.871,155.862
C07869=1049.578,-116.702,-67.647,169.812,30.871,155.862
C07870=1049.572,-116.952,-67.637,169.810,30.870,155.862
C07871=1049.566,-117.202,-67.628,169.808,30.870,155.862
C07872=1049.560,-117.451,-67.618,169.806,30.870,155.862
C07873=1049.554,-117.701,-67.608,169.804,30.869,155.862
C07874=1049.548,-117.951,-67.599,169.802,30.869,155.863
C07875=1049.542,-118.200,-67.590,169.800,30.869,155.863
C07876=1049.536,-118.450,-67.581,169.798,30.868,155.863
C07877=1049.529,-118.700,-67.572,169.795,30.868,155.863
C07878=1049.523,-118.950,-67.562,169.793,30.868,155.863
C07879=1049.517,-119.200,-67.553,169.791,30.868,155.863
C07880=1049.511,-119.449,-67.543,169.789,30.868,155.863
C07881=1049.505,-119.699,-67.534,169.786,30.867,155.863
C07882=1049.498,-119.949,-67.524,169.784,30.867,155.863
C07883=1049.493,-120.198,-67.515,169.782,30.867,155.863
C07884=1049.487,-120.448,-67.506,169.780,30.866,155.863
C07885=1049.481,-120.698,-67.496,169.777,30.866,155.863
C07886=1049.474,-120.948,-67.487,169.775,30.866,155.864
C07887=1049.468,-121.198,-67.478,169.773,30.865,155.864
C07888=1049.462,-121.447,-67.469,169.771,30.865,155.864
C07889=1049.456,-121.697,-67.460,169.769,30.864,155.864
C07890=1049.450,-121.947,-67.450,169.767,30.865,155.864
C07891=1049.444,-122.197,-67.441,169.765,30.864,155.864
C07892=1049.437,-122.446,-67.432,169.763,30.864,155.864
C07893=1049.431,-122.697,-67.423,169.760,30.864,155.864
C07894=1049.426,-122.946,-67.414,169.758,30.863,155.864
C07895=1049.419,-123.195,-67.404,169.756,30.863,155.864
C07896=1049.413,-123.445,-67.394,169.754,30.863,155.864
C07897=1049.407,-123.696,-67.386,169.751,30.863,155.865
C07898=1049.401,-123.944,-67.377,169.749,30.863,155.865
C07899=1049.395,-124.194,-67.367,169.747,30.862,155.865
C07900=1049.389,-124.444,-67.358,169.744,30.862,155.865
C07901=1049.383,-124.694,-67.349,169.742,30.862,155.865
C07902=1049.376,-124.944,-67.340,169.740,30.862,155.865
C07903=1049.370,-125.193,-67.331,169.738,30.862,155.865
C07904=1049.364,-125.443,-67.322,169.735,30.861,155.865
C07905=1049.358,-125.693,-67.312,169.733,30.861,155.865
C07906=1049.351,-125.943,-67.303,169.732,30.861,155.865
C07907=1049.346,-126.192,-67.295,169.730,30.861,155.865
C07908=1049.340,-126.442,-67.285,169.727,30.860,155.866
C07909=1049.333,-126.692,-67.277,169.725,30.861,155.866
C07910=1049.327,-126.942,-67.268,169.723,30.860,155.866
C07911=1049.322,-127.191,-67.258,169.721,30.860,155.866
C07912=1049.315,-127.441,-67.250,169.718,30.860,155.866
C07913=1049.309,-127.691,-67.241,169.716,30.860,155.866
C07914=1049.303,-127.940,-67.231,169.714,30.860,155.866
C07915=1049.299,-128.190,-67.222,169.712,30.859,155.866
C07916=1049.295,-128.440,-67.211,169.710,30.858,155.866
C07917=1049.292,-128.690,-67.200,169.708,30.856,155.866
C07918=1049.291,-128.940,-67.189,169.706,30.853,155.866
C07919=1049.290,-129.191,-67.176,169.705,30.851,155.865
C07920=1049.290,-129.441,-67.163,169.703,30.847,155.865
C07921=1049.293,-129.692,-67.149,169.702,30.844,155.864
C07922=1049.295,-129.942,-67.135,169.700,30.840,155.864
C07923=1049.298,-130.193,-67.120,169.700,30.835,155.863
C07924=1049.302,-130.443,-67.104,169.699,30.830,155.862
C07925=1049.307,-130.694,-67.087,169.698,30.824,155.861
C07926=1049.314,-130.944,-67.071,169.698,30.819,155.860
C07927=1048.952,-130.967,-67.300,169.651,30.989,155.892
C07928=1048.945,-130.717,-67.316,169.652,30.995,155.893
C07929=1048.940,-130.467,-67.333,169.653,31.000,155.894
C07930=1048.935,-130.216,-67.348,169.654,31.006,155.895
C07931=1048.932,-129.965,-67.364,169.655,31.010,155.896
C07932=1048.929,-129.715,-67.377,169.656,31.015,155.896
C07933=1048.928,-129.465,-67.392,169.658,31.018,155.897
C07934=1048.927,-129.215,-67.405,169.659,31.022,155.897
C07935=1048.928,-128.964,-67.418,169.660,31.024,155.898
C07936=1048.930,-128.714,-67.429,169.662,31.027,155.898
C07937=1048.932,-128.464,-67.440,169.664,31.028,155.898
C07938=1048.935,-128.214,-67.450,169.666,31.030,155.898
C07939=1048.940,-127.964,-67.460,169.668,31.031,155.898
C07940=1048.946,-127.715,-67.470,169.670,31.031,155.898
C07941=1048.952,-127.465,-67.479,169.673,31.031,155.898
C07942=1048.958,-127.215,-67.488,169.675,31.031,155.898
C07943=1048.964,-126.966,-67.497,169.677,31.031,155.898
C07944=1048.970,-126.715,-67.506,169.679,31.031,155.898
C07945=1048.976,-126.466,-67.515,169.681,31.031,155.898
C07946=1048.983,-126.217,-67.524,169.683,31.032,155.898
C07947=1048.989,-125.966,-67.533,169.685,31.031,155.897
C07948=1048.995,-125.716,-67.542,169.688,31.032,155.897
C07949=1049.001,-125.468,-67.551,169.690,31.032,155.897
C07950=1049.007,-125.217,-67.560,169.692,31.032,155.897
C07951=1049.013,-124.967,-67.569,169.695,31.032,155.897
C07952=1049.019,-124.718,-67.579,169.697,31.033,155.897
C07953=1049.026,-124.467,-67.587,169.699,31.033,155.897
C07954=1049.032,-124.218,-67.596,169.701,31.032,155.897
C07955=1049.038,-123.969,-67.606,169.704,31.033,155.897
C07956=1049.044,-123.718,-67.615,169.706,31.033,155.897
C07957=1049.050,-123.469,-67.624,169.708,31.034,155.897
C07958=1049.056,-123.220,-67.633,169.710,31.034,155.896
C07959=1049.062,-122.970,-67.642,169.713,31.034,155.896
C07960=1049.068,-122.719,-67.651,169.715,31.034,155.896
C07961=1049.074,-122.470,-67.661,169.717,31.034,155.896
C07962=1049.080,-122.220,-67.670,169.719,31.035,155.896
C07963=1049.087,-121.971,-67.679,169.721,31.035,155.896
C07964=1049.093,-121.721,-67.688,169.723,31.035,155.896
C07965=1049.099,-121.471,-67.697,169.725,31.036,155.896
C07966=1049.105,-121.221,-67.707,169.728,31.035,155.896
C07967=1049.111,-120.971,-67.716,169.730,31.036,155.896
C07968=1049.117,-120.722,-67.726,169.732,31.036,155.896
C07969=1049.123,-120.472,-67.735,169.734,31.036,155.895
C07970=1049.129,-120.222,-67.744,169.737,31.037,155.895
C07971=1049.136,-119.972,-67.753,169.739,31.037,155.895
C07972=1049.142,-119.723,-67.763,169.741,31.037,155.895
C07973=1049.148,-119.473,-67.772,169.743,31.038,155.895
C07974=1049.154,-119.223,-67.782,169.746,31.038,155.895
C07975=1049.160,-118.974,-67.791,169.748,31.038,155.895
C07976=1049.166,-118.723,-67.800,169.750,31.039,155.895
C07977=1049.172,-118.474,-67.809,169.752,31.038,155.895
C07978=1049.178,-118.224,-67.819,169.755,31.039,155.895
C07979=1049.185,-117.974,-67.828,169.756,31.039,155.895
C07980=1049.191,-117.725,-67.838,169.758,31.039,155.895
C07981=1049.197,-117.475,-67.847,169.761,31.040,155.894
C07982=1049.203,-117.225,-67.857,169.763,31.040,155.894
C07983=1049.209,-116.976,-67.866,169.765,31.040,155.894
C07984=1049.215,-116.726,-67.875,169.767,31.041,155.894
C07985=1049.221,-116.476,-67.885,169.770,31.041,155.894
C07986=1049.227,-116.227,-67.895,169.772,31.041,155.894
C07987=1049.234,-115.977,-67.904,169.774,31.042,155.894
C07988=1049.241,-115.692,-67.915,169.777,31.042,155.894
C07989=1049.247,-115.406,-67.925,169.779,31.043,155.894
C07990=1049.255,-115.120,-67.936,169.782,31.043,155.894
C07991=1049.262,-114.835,-67.947,169.784,31.044,155.894
C07992=1049.268,-114.585,-67.956,169.787,31.044,155.894
C07993=1049.274,-114.336,-67.966,169.789,31.045,155.894
C07994=1049.280,-114.086,-67.976,169.790,31.045,155.894
C07995=1049.286,-113.836,-67.985,169.792,31.045,155.894
C07996=1049.292,-113.587,-67.996,169.795,31.046,155.893
C07997=1049.298,-113.337,-68.006,169.797,31.046,155.893
C07998=1049.304,-113.088,-68.015,169.799,31.046,155.893
C07999=1049.310,-112.838,-68.024,169.801,31.047,155.893
C08000=1049.316,-112.588,-68.034,169.804,31.048,155.893
C08001=1049.322,-112.338,-68.043,169.806,31.048,155.893
C08002=1049.329,-112.088,-68.053,169.808,31.048,155.893
C08003=1049.335,-111.839,-68.063,169.810,31.049,155.893
C08004=1049.341,-111.589,-68.072,169.813,31.049,155.893
C08005=1049.347,-111.339,-68.082,169.815,31.049,155.893
C08006=1049.354,-111.090,-68.092,169.817,31.050,155.893
C08007=1049.360,-110.840,-68.102,169.819,31.050,155.893
C08008=1049.365,-110.590,-68.112,169.822,31.051,155.893
C08009=1049.371,-110.340,-68.121,169.823,31.051,155.893
C08010=1049.378,-110.090,-68.131,169.825,31.052,155.893
C08011=1049.384,-109.841,-68.140,169.827,31.052,155.893
C08012=1049.390,-109.591,-68.151,169.830,31.053,155.893
C08013=1049.396,-109.342,-68.160,169.832,31.053,155.893
C08014=1049.403,-109.092,-68.170,169.834,31.053,155.893
C08015=1049.409,-108.842,-68.179,169.836,31.054,155.893
C08016=1049.415,-108.592,-68.189,169.839,31.055,155.893
C08017=1049.421,-108.343,-68.200,169.841,31.055,155.892
C08018=1049.427,-108.093,-68.209,169.843,31.055,155.892
C08019=1049.433,-107.843,-68.219,169.845,31.056,155.892
C08020=1049.440,-107.593,-68.229,169.848,31.057,155.892
C08021=1049.446,-107.343,-68.239,169.850,31.057,155.892
C08022=1049.452,-107.094,-68.249,169.852,31.057,155.892
C08023=1049.458,-106.844,-68.259,169.853,31.058,155.892
C08024=1049.464,-106.594,-68.269,169.855,31.059,155.892
C08025=1049.470,-106.345,-68.279,169.858,31.059,155.892
C08026=1049.477,-106.095,-68.288,169.860,31.060,155.892
C08027=1049.482,-105.845,-68.299,169.862,31.060,155.892
C08028=1049.489,-105.595,-68.309,169.864,31.061,155.892
C08029=1049.495,-105.346,-68.318,169.867,31.062,155.892
C08030=1049.501,-105.096,-68.328,169.869,31.062,155.892
C08031=1049.507,-104.846,-68.339,169.871,31.063,155.892
C08032=1049.513,-104.597,-68.348,169.873,31.063,155.892
C08033=1049.519,-104.347,-68.358,169.876,31.064,155.892
C08034=1049.525,-104.098,-68.368,169.878,31.065,155.892
C08035=1049.532,-103.847,-68.379,169.880,31.065,155.892
C08036=1049.538,-103.597,-68.388,169.882,31.066,155.892
C08037=1049.544,-103.348,-68.399,169.883,31.066,155.892
C08038=1049.550,-103.098,-68.409,169.886,31.066,155.892
C08039=1049.556,-102.849,-68.419,169.888,31.067,155.892
C08040=1049.562,-102.599,-68.429,169.890,31.068,155.892
C08041=1049.568,-102.349,-68.440,169.892,31.069,155.892
C08042=1049.574,-102.099,-68.449,169.895,31.069,155.892
C08043=1049.580,-101.850,-68.459,169.897,31.070,155.892
C08044=1049.587,-101.599,-68.470,169.899,31.070,155.892
C08045=1049.593,-101.350,-68.479,169.901,31.071,155.892
C08046=1049.599,-101.101,-68.490,169.903,31.071,155.892
C08047=1049.605,-100.850,-68.500,169.906,31.073,155.892
C08048=1049.611,-100.601,-68.510,169.908,31.073,155.892
C08049=1049.617,-100.351,-68.520,169.910,31.074,155.892
C08050=1049.624,-100.101,-68.531,169.911,31.074,155.892
C08051=1049.630,-99.851,-68.541,169.914,31.075,155.892
C08052=1049.637,-99.565,-68.552,169.916,31.075,155.892
C08053=1049.644,-99.279,-68.564,169.919,31.076,155.892
C08054=1049.652,-98.993,-68.576,169.921,31.077,155.892
C08055=1049.658,-98.706,-68.588,169.924,31.078,155.892
C08056=1049.665,-98.456,-68.598,169.926,31.079,155.892
C08057=1049.671,-98.207,-68.608,169.928,31.079,155.892
C08058=1049.677,-97.957,-68.618,169.930,31.080,155.892
C08059=1049.683,-97.708,-68.629,169.933,31.080,155.892
C08060=1049.689,-97.458,-68.639,169.935,31.081,155.892
C08061=1049.696,-97.208,-68.649,169.937,31.082,155.892
C08062=1049.701,-96.958,-68.660,169.938,31.083,155.892
C08063=1049.707,-96.708,-68.670,169.940,31.083,155.892
C08064=1049.713,-96.459,-68.681,169.943,31.085,155.892
C08065=1049.720,-96.210,-68.691,169.945,31.085,155.892
C08066=1049.726,-95.959,-68.701,169.947,31.086,155.892
C08067=1049.732,-95.710,-68.712,169.949,31.087,155.892
C08068=1049.738,-95.460,-68.723,169.951,31.087,155.892
C08069=1049.743,-95.210,-68.733,169.954,31.088,155.892
C08070=1049.750,-94.961,-68.743,169.956,31.089,155.892
C08071=1049.756,-94.711,-68.754,169.958,31.090,155.892
C08072=1049.763,-94.461,-68.765,169.960,31.090,155.892
C08073=1049.768,-94.211,-68.775,169.962,31.091,155.892
C08074=1049.774,-93.962,-68.786,169.964,31.092,155.892
C08075=1049.780,-93.713,-68.796,169.966,31.093,155.892
C08076=1049.787,-93.462,-68.807,169.968,31.093,155.892
C08077=1049.792,-93.212,-68.817,169.970,31.094,155.892
C08078=1049.799,-92.963,-68.828,169.972,31.095,155.892
C08079=1049.804,-92.714,-68.838,169.974,31.096,155.892
C08080=1049.811,-92.464,-68.849,169.977,31.097,155.892
C08081=1049.817,-92.214,-68.859,169.979,31.097,155.892
C08082=1049.823,-91.964,-68.870,169.981,31.098,155.892
C08083=1049.830,-91.714,-68.881,169.983,31.099,155.892
C08084=1049.835,-91.465,-68.892,169.985,31.100,155.892
C08085=1049.842,-91.216,-68.902,169.987,31.101,155.892
C08086=1049.847,-90.966,-68.912,169.989,31.102,155.892
C08087=1049.854,-90.715,-68.923,169.991,31.103,155.892
C08088=1049.860,-90.466,-68.934,169.993,31.103,155.892
C08089=1049.866,-90.217,-68.945,169.995,31.104,155.892
C08090=1049.872,-89.966,-68.956,169.998,31.105,155.892
C08091=1049.879,-89.717,-68.966,170.000,31.106,155.892
C08092=1049.884,-89.468,-68.977,170.002,31.107,155.892
C08093=1049.890,-89.217,-68.987,170.004,31.108,155.892
C08094=1049.897,-88.968,-68.998,170.006,31.108,155.892
C08095=1049.903,-88.718,-69.009,170.008,31.109,155.892
C08096=1049.909,-88.468,-69.020,170.011,31.110,155.892
C08097=1049.915,-88.219,-69.030,170.012,31.111,155.892
C08098=1049.921,-87.969,-69.041,170.014,31.112,155.892
C08099=1049.928,-87.719,-69.052,170.016,31.113,155.892
C08100=1049.934,-87.470,-69.063,170.018,31.113,155.892
C08101=1049.940,-87.220,-69.074,170.021,31.115,155.892
C08102=1049.946,-86.970,-69.085,170.023,31.115,155.892
C08103=1049.953,-86.721,-69.095,170.025,31.116,155.892
C08104=1049.959,-86.471,-69.106,170.027,31.117,155.893
C08105=1049.965,-86.222,-69.117,170.029,31.118,155.893
C08106=1049.971,-85.972,-69.127,170.031,31.119,155.893
C08107=1049.977,-85.722,-69.139,170.034,31.120,155.893
C08108=1049.983,-85.473,-69.149,170.036,31.120,155.893
C08109=1049.990,-85.223,-69.160,170.037,31.121,155.893
C08110=1049.996,-84.973,-69.171,170.039,31.122,155.893
C08111=1050.002,-84.723,-69.182,170.041,31.123,155.893
C08112=1050.009,-84.474,-69.193,170.043,31.124,155.893
C08113=1050.015,-84.224,-69.203,170.046,31.125,155.893
C08114=1050.021,-83.974,-69.215,170.048,31.126,155.893
C08115=1050.027,-83.725,-69.226,170.050,31.127,155.893
C08116=1050.034,-83.441,-69.238,170.052,31.128,155.893
C08117=1050.041,-83.156,-69.250,170.055,31.129,155.893
C08118=1050.049,-82.872,-69.263,170.057,31.130,155.893
C08119=1050.056,-82.588,-69.275,170.059,31.131,155.893
C08120=1050.062,-82.338,-69.286,170.061,31.132,155.893
C08121=1050.069,-82.088,-69.297,170.063,31.133,155.893
C08122=1050.074,-81.839,-69.308,170.065,31.134,155.893
C08123=1050.081,-81.589,-69.319,170.068,31.135,155.893
C08124=1050.087,-81.340,-69.330,170.070,31.136,155.893
C08125=1050.094,-81.090,-69.341,170.072,31.137,155.893
C08126=1050.100,-80.840,-69.352,170.074,31.138,155.893
C08127=1050.106,-80.590,-69.363,170.076,31.138,155.893
C08128=1050.112,-80.341,-69.374,170.078,31.139,155.893
C08129=1050.119,-80.091,-69.385,170.080,31.140,155.894
C08130=1050.125,-79.842,-69.396,170.082,31.141,155.894
C08131=1050.131,-79.592,-69.408,170.084,31.142,155.894
C08132=1050.137,-79.342,-69.418,170.086,31.144,155.894
C08133=1050.143,-79.092,-69.430,170.088,31.145,155.894
C08134=1050.149,-78.843,-69.441,170.090,31.146,155.894
C08135=1050.156,-78.593,-69.453,170.092,31.147,155.894
C08136=1050.161,-78.344,-69.463,170.095,31.148,155.894
C08137=1050.168,-78.093,-69.475,170.097,31.149,155.894
C08138=1050.173,-77.844,-69.486,170.099,31.150,155.894
C08139=1050.180,-77.594,-69.497,170.101,31.151,155.894
C08140=1050.187,-77.345,-69.508,170.103,31.152,155.894
C08141=1050.193,-77.095,-69.519,170.104,31.153,155.894
C08142=1050.199,-76.846,-69.531,170.106,31.154,155.894
C08143=1050.205,-76.596,-69.542,170.108,31.155,155.895
C08144=1050.211,-76.346,-69.553,170.111,31.156,155.895
C08145=1050.218,-76.097,-69.565,170.113,31.157,155.895
C08146=1050.223,-75.847,-69.576,170.115,31.158,155.895
C08147=1050.230,-75.597,-69.587,170.117,31.159,155.895
C08148=1050.236,-75.348,-69.599,170.119,31.161,155.895
C08149=1050.242,-75.098,-69.610,170.121,31.161,155.895
C08150=1050.248,-74.848,-69.621,170.123,31.162,155.895
C08151=1050.254,-74.599,-69.632,170.125,31.163,155.895
C08152=1050.261,-74.349,-69.644,170.127,31.165,155.895
C08153=1050.267,-74.100,-69.655,170.129,31.166,155.895
C08154=1050.273,-73.850,-69.667,170.131,31.167,155.895
C08155=1050.279,-73.599,-69.678,170.133,31.168,155.895
C08156=1050.285,-73.350,-69.690,170.135,31.169,155.895
C08157=1050.291,-73.100,-69.701,170.137,31.170,155.896
C08158=1050.297,-72.851,-69.713,170.139,31.172,155.896
C08159=1050.304,-72.601,-69.724,170.142,31.173,155.896
C08160=1050.309,-72.352,-69.736,170.144,31.174,155.896
C08161=1050.315,-72.102,-69.748,170.145,31.175,155.896
C08162=1050.321,-71.853,-69.759,170.147,31.176,155.896
C08163=1050.328,-71.603,-69.770,170.149,31.178,155.896
C08164=1050.334,-71.353,-69.783,170.151,31.179,155.896
C08165=1050.339,-71.103,-69.794,170.153,31.180,155.896
C08166=1050.346,-70.854,-69.806,170.155,31.181,155.896
C08167=1050.352,-70.604,-69.817,170.157,31.183,155.897
C08168=1050.358,-70.354,-69.829,170.159,31.183,155.897
C08169=1050.363,-70.105,-69.840,170.162,31.184,155.897
C08170=1050.370,-69.855,-69.852,170.164,31.186,155.897
C08171=1050.376,-69.605,-69.863,170.165,31.187,155.897
C08172=1050.382,-69.356,-69.875,170.167,31.188,155.897
C08173=1050.388,-69.106,-69.887,170.169,31.189,155.897
C08174=1050.395,-68.856,-69.899,170.171,31.191,155.897
C08175=1050.401,-68.607,-69.910,170.173,31.192,155.897
C08176=1050.406,-68.357,-69.922,170.175,31.193,155.897
C08177=1050.413,-68.107,-69.934,170.177,31.194,155.897
C08178=1050.419,-67.858,-69.946,170.179,31.196,155.898
C08179=1050.425,-67.608,-69.957,170.182,31.197,155.898
C08180=1050.432,-67.326,-69.971,170.184,31.198,155.898
C08181=1050.439,-67.045,-69.984,170.185,31.200,155.898
C08182=1050.445,-66.762,-69.997,170.188,31.201,155.898
C08183=1050.453,-66.480,-70.011,170.190,31.202,155.898
C08184=1050.459,-66.231,-70.022,170.192,31.203,155.898
C08185=1050.465,-65.981,-70.033,170.194,31.205,155.898
C08186=1050.471,-65.731,-70.046,170.196,31.206,155.899
C08187=1050.477,-65.482,-70.058,170.198,31.207,155.899
C08188=1050.483,-65.232,-70.069,170.200,31.209,155.899
C08189=1050.490,-64.983,-70.081,170.203,31.210,155.899
C08190=1050.496,-64.733,-70.093,170.204,31.211,155.899
C08191=1050.502,-64.484,-70.105,170.206,31.212,155.899
C08192=1050.508,-64.234,-70.116,170.208,31.214,155.899
C08193=1050.514,-63.984,-70.129,170.210,31.215,155.899
C08194=1050.520,-63.735,-70.140,170.212,31.216,155.899
C08195=1050.527,-63.485,-70.152,170.214,31.217,155.899
C08196=1050.532,-63.235,-70.164,170.216,31.219,155.900
C08197=1050.539,-62.985,-70.176,170.218,31.220,155.900
C08198=1050.545,-62.736,-70.188,170.220,31.221,155.900
C08199=1050.551,-62.486,-70.200,170.222,31.223,155.900
C08200=1050.558,-62.237,-70.212,170.224,31.224,155.900
C08201=1050.564,-61.987,-70.223,170.226,31.225,155.900
C08202=1050.570,-61.737,-70.236,170.228,31.226,155.900
C08203=1050.576,-61.488,-70.248,170.230,31.228,155.900
C08204=1050.583,-61.238,-70.260,170.232,31.229,155.900
C08205=1050.588,-60.988,-70.272,170.234,31.230,155.901
C08206=1050.595,-60.739,-70.284,170.236,31.232,155.901
C08207=1050.601,-60.489,-70.295,170.238,31.233,155.901
C08208=1050.607,-60.239,-70.308,170.240,31.234,155.901
C08209=1050.613,-59.990,-70.319,170.242,31.235,155.901
C08210=1050.620,-59.740,-70.331,170.243,31.237,155.901
C08211=1050.626,-59.490,-70.344,170.245,31.238,155.901
C08212=1050.633,-59.241,-70.356,170.247,31.239,155.901
C08213=1050.639,-58.992,-70.368,170.249,31.240,155.902
C08214=1050.645,-58.742,-70.380,170.252,31.242,155.902
C08215=1050.651,-58.493,-70.392,170.254,31.243,155.902
C08216=1050.657,-58.242,-70.404,170.256,31.245,155.902
C08217=1050.663,-57.992,-70.416,170.258,31.245,155.902
C08218=1050.670,-57.743,-70.428,170.260,31.247,155.902
C08219=1050.676,-57.493,-70.440,170.261,31.249,155.902
C08220=1050.683,-57.243,-70.452,170.263,31.249,155.902
C08221=1050.689,-56.995,-70.464,170.265,31.251,155.903
C08222=1050.695,-56.745,-70.476,170.267,31.252,155.903
C08223=1050.701,-56.495,-70.488,170.269,31.253,155.903
C08224=1050.707,-56.245,-70.501,170.271,31.255,155.903
C08225=1050.714,-55.996,-70.513,170.273,31.256,155.903
C08226=1050.720,-55.746,-70.525,170.275,31.257,155.903
C08227=1050.726,-55.496,-70.537,170.277,31.259,155.903
C08228=1050.733,-55.247,-70.549,170.279,31.260,155.903
C08229=1050.740,-54.997,-70.561,170.281,31.261,155.904
C08230=1050.746,-54.747,-70.574,170.283,31.263,155.904
C08231=1050.752,-54.498,-70.586,170.285,31.264,155.904
C08232=1050.758,-54.248,-70.598,170.287,31.265,155.904
C08233=1050.764,-54.000,-70.611,170.289,31.267,155.904
C08234=1050.770,-53.750,-70.623,170.291,31.268,155.904
C08235=1050.777,-53.500,-70.635,170.293,31.269,155.904
C08236=1050.784,-53.250,-70.647,170.295,31.271,155.904
C08237=1050.790,-53.001,-70.660,170.297,31.272,155.905
C08238=1050.796,-52.751,-70.672,170.299,31.273,155.905
C08239=1050.802,-52.501,-70.684,170.300,31.275,155.905
C08240=1050.809,-52.252,-70.696,170.302,31.276,155.905
C08241=1050.815,-52.002,-70.708,170.304,31.277,155.905
C08242=1050.821,-51.752,-70.721,170.306,31.279,155.905
C08243=1050.828,-51.503,-70.733,170.308,31.280,155.905
C08244=1050.835,-51.222,-70.747,170.311,31.282,155.906
C08245=1050.843,-50.942,-70.761,170.313,31.283,155.906
C08246=1050.849,-50.661,-70.775,170.315,31.285,155.906
C08247=1050.857,-50.380,-70.789,170.318,31.287,155.906
C08248=1050.863,-50.130,-70.801,170.319,31.288,155.906
C08249=1050.869,-49.880,-70.814,170.321,31.289,155.906
C08250=1050.875,-49.631,-70.826,170.323,31.291,155.906
C08251=1050.881,-49.382,-70.839,170.325,31.292,155.907
C08252=1050.887,-49.132,-70.851,170.327,31.294,155.907
C08253=1050.893,-48.883,-70.864,170.329,31.295,155.907
C08254=1050.899,-48.633,-70.876,170.331,31.297,155.907
C08255=1050.905,-48.383,-70.890,170.333,31.298,155.907
C08256=1050.912,-48.134,-70.902,170.335,31.300,155.907
C08257=1050.918,-47.884,-70.914,170.336,31.301,155.908
C08258=1050.924,-47.635,-70.928,170.338,31.303,155.908
C08259=1050.930,-47.385,-70.940,170.340,31.304,155.908
C08260=1050.937,-47.135,-70.952,170.342,31.306,155.908
C08261=1050.943,-46.886,-70.965,170.344,31.307,155.908
C08262=1050.949,-46.636,-70.978,170.346,31.309,155.908
C08263=1050.955,-46.386,-70.990,170.348,31.310,155.909
C08264=1050.962,-46.137,-71.003,170.350,31.312,155.909
C08265=1050.968,-45.887,-71.016,170.352,31.313,155.909
C08266=1050.974,-45.638,-71.028,170.353,31.315,155.909
C08267=1050.980,-45.388,-71.041,170.355,31.316,155.909
C08268=1050.986,-45.139,-71.053,170.357,31.318,155.909
C08269=1050.993,-44.889,-71.067,170.359,31.319,155.910
C08270=1050.999,-44.640,-71.079,170.361,31.321,155.910
C08271=1051.004,-44.390,-71.092,170.363,31.322,155.910
C08272=1051.011,-44.140,-71.105,170.365,31.324,155.910
C08273=1051.017,-43.891,-71.117,170.367,31.325,155.910
C08274=1051.024,-43.641,-71.131,170.369,31.327,155.910
C08275=1051.030,-43.391,-71.143,170.371,31.329,155.911
C08276=1051.036,-43.142,-71.157,170.372,31.330,155.911
C08277=1051.042,-42.892,-71.169,170.374,31.332,155.911
C08278=1051.049,-42.642,-71.181,170.376,31.333,155.911
C08279=1051.055,-42.393,-71.194,170.378,31.335,155.911
C08280=1051.061,-42.143,-71.207,170.380,31.336,155.911
C08281=1051.067,-41.894,-71.220,170.382,31.338,155.912
C08282=1051.073,-41.644,-71.233,170.384,31.339,155.912
C08283=1051.079,-41.395,-71.246,170.386,31.341,155.912
C08284=1051.086,-41.145,-71.258,170.388,31.342,155.912
C08285=1051.093,-40.895,-71.272,170.389,31.344,155.912
C08286=1051.099,-40.645,-71.284,170.391,31.345,155.912
C08287=1051.105,-40.396,-71.297,170.393,31.347,155.913
C08288=1051.111,-40.147,-71.311,170.395,31.348,155.913
C08289=1051.118,-39.897,-71.323,170.397,31.350,155.913
C08290=1051.124,-39.648,-71.336,170.399,31.351,155.913
C08291=1051.130,-39.398,-71.348,170.401,31.353,155.913
C08292=1051.137,-39.148,-71.362,170.403,31.354,155.913
C08293=1051.143,-38.898,-71.375,170.405,31.356,155.914
C08294=1051.149,-38.649,-71.388,170.406,31.357,155.914
C08295=1051.155,-38.400,-71.401,170.408,31.359,155.914
C08296=1051.161,-38.150,-71.414,170.410,31.361,155.914
C08297=1051.167,-37.900,-71.427,170.412,31.362,155.914
C08298=1051.173,-37.651,-71.440,170.414,31.364,155.915
C08299=1051.180,-37.401,-71.453,170.415,31.365,155.915
C08300=1051.186,-37.151,-71.466,170.417,31.367,155.915
C08301=1051.192,-36.902,-71.480,170.419,31.369,155.915
C08302=1051.198,-36.652,-71.492,170.421,31.370,155.915
C08303=1051.204,-36.403,-71.506,170.422,31.372,155.916
C08304=1051.211,-36.154,-71.519,170.424,31.374,155.916
C08305=1051.216,-35.904,-71.531,170.426,31.375,155.916
C08306=1051.223,-35.654,-71.545,170.428,31.377,155.916
C08307=1051.230,-35.405,-71.558,170.430,31.379,155.916
C08308=1051.237,-35.125,-71.573,170.432,31.380,155.916
C08309=1051.243,-34.844,-71.588,170.435,31.382,155.917
C08310=1051.250,-34.563,-71.602,170.437,31.384,155.917
C08311=1051.257,-34.283,-71.617,170.439,31.386,155.917
C08312=1051.263,-34.034,-71.630,170.440,31.388,155.917
C08313=1051.269,-33.785,-71.644,170.442,31.389,155.917
C08314=1051.276,-33.535,-71.657,170.444,31.391,155.918
C08315=1051.282,-33.285,-71.670,170.446,31.393,155.918
C08316=1051.288,-33.036,-71.683,170.448,31.394,155.918
C08317=1051.294,-32.786,-71.696,170.450,31.396,155.918
C08318=1051.300,-32.537,-71.710,170.452,31.397,155.918
C08319=1051.307,-32.287,-71.724,170.454,31.399,155.919
C08320=1051.313,-32.038,-71.737,170.455,31.401,155.919
C08321=1051.319,-31.788,-71.750,170.456,31.402,155.919
C08322=1051.325,-31.538,-71.763,170.458,31.404,155.919
C08323=1051.332,-31.288,-71.777,170.460,31.406,155.920
C08324=1051.338,-31.039,-71.790,170.462,31.407,155.920
C08325=1051.344,-30.790,-71.803,170.464,31.409,155.920
C08326=1051.350,-30.541,-71.817,170.466,31.410,155.920
C08327=1051.357,-30.291,-71.830,170.468,31.413,155.920
C08328=1051.362,-30.041,-71.843,170.470,31.414,155.921
C08329=1051.369,-29.791,-71.857,170.472,31.416,155.921
C08330=1051.375,-29.541,-71.870,170.473,31.417,155.921
C08331=1051.382,-29.292,-71.883,170.475,31.419,155.921
C08332=1051.388,-29.043,-71.897,170.477,31.421,155.921
C08333=1051.395,-28.793,-71.910,170.479,31.422,155.921
C08334=1051.401,-28.544,-71.924,170.481,31.424,155.922
C08335=1051.407,-28.294,-71.937,170.483,31.426,155.922
C08336=1051.413,-28.045,-71.951,170.485,31.427,155.922
C08337=1051.419,-27.795,-71.964,170.486,31.429,155.922
C08338=1051.426,-27.546,-71.978,170.488,31.431,155.923
C08339=1051.432,-27.296,-71.991,170.489,31.432,155.923
C08340=1051.439,-27.046,-72.005,170.491,31.434,155.923
C08341=1051.445,-26.797,-72.018,170.493,31.435,155.923
C08342=1051.450,-26.547,-72.032,170.495,31.437,155.923
C08343=1051.457,-26.297,-72.045,170.497,31.439,155.924
C08344=1051.463,-26.048,-72.059,170.499,31.441,155.924
C08345=1051.469,-25.799,-72.073,170.501,31.443,155.924
C08346=1051.476,-25.549,-72.086,170.503,31.445,155.924
C08347=1051.481,-25.299,-72.100,170.505,31.446,155.924
C08348=1051.487,-25.050,-72.113,170.506,31.448,155.925
C08349=1051.494,-24.800,-72.127,170.507,31.450,155.925
C08350=1051.500,-24.550,-72.141,170.509,31.451,155.925
C08351=1051.506,-24.301,-72.154,170.511,31.453,155.925
C08352=1051.513,-24.051,-72.168,170.513,31.455,155.926
C08353=1051.518,-23.802,-72.182,170.515,31.457,155.926
C08354=1051.525,-23.553,-72.196,170.517,31.458,155.926
C08355=1051.531,-23.303,-72.209,170.519,31.460,155.926
C08356=1051.537,-23.053,-72.223,170.521,31.462,155.926
C08357=1051.543,-22.804,-72.236,170.523,31.464,155.927
C08358=1051.549,-22.554,-72.251,170.524,31.466,155.927
C08359=1051.555,-22.304,-72.264,170.525,31.467,155.927
C08360=1051.563,-22.055,-72.278,170.527,31.469,155.927
C08361=1051.568,-21.806,-72.292,170.529,31.471,155.928
C08362=1051.574,-21.556,-72.305,170.531,31.473,155.928
C08363=1051.580,-21.306,-72.320,170.533,31.474,155.928
C08364=1051.587,-21.057,-72.333,170.535,31.476,155.928
C08365=1051.594,-20.807,-72.347,170.537,31.478,155.928
C08366=1051.599,-20.558,-72.361,170.539,31.479,155.929
C08367=1051.605,-20.309,-72.374,170.540,31.482,155.929
C08368=1051.611,-20.058,-72.389,170.542,31.483,155.929
C08369=1051.618,-19.809,-72.402,170.543,31.485,155.929
C08370=1051.625,-19.560,-72.416,170.545,31.487,155.930
C08371=1051.630,-19.310,-72.430,170.547,31.489,155.930
C08372=1051.637,-19.029,-72.446,170.549,31.490,155.930
C08373=1051.645,-18.748,-72.461,170.551,31.492,155.930
C08374=1051.652,-18.467,-72.477,170.554,31.495,155.931
C08375=1051.659,-18.186,-72.492,170.555,31.497,155.931
C08376=1051.665,-17.937,-72.506,170.557,31.498,155.931
C08377=1051.671,-17.687,-72.521,170.558,31.500,155.931
C08378=1051.678,-17.438,-72.534,170.560,31.502,155.931
C08379=1051.684,-17.188,-72.548,170.562,31.504,155.932
C08380=1051.690,-16.939,-72.562,170.564,31.505,155.932
C08381=1051.696,-16.689,-72.576,170.566,31.507,155.932
C08382=1051.702,-16.439,-72.590,170.568,31.509,155.932
C08383=1051.709,-16.190,-72.605,170.570,31.511,155.933
C08384=1051.715,-15.940,-72.618,170.572,31.512,155.933
C08385=1051.722,-15.690,-72.631,170.573,31.515,155.933
C08386=1051.728,-15.442,-72.646,170.574,31.516,155.933
C08387=1051.734,-15.192,-72.660,170.576,31.518,155.934
C08388=1051.740,-14.943,-72.674,170.578,31.520,155.934
C08389=1051.746,-14.692,-72.688,170.580,31.522,155.934
C08390=1051.752,-14.443,-72.702,170.582,31.523,155.934
C08391=1051.759,-14.193,-72.717,170.584,31.525,155.935
C08392=1051.764,-13.944,-72.731,170.586,31.527,155.935
C08393=1051.771,-13.694,-72.745,170.587,31.529,155.935
C08394=1051.777,-13.445,-72.759,170.588,31.531,155.935
C08395=1051.783,-13.195,-72.774,170.590,31.533,155.936
C08396=1051.790,-12.946,-72.787,170.592,31.534,155.936
C08397=1051.796,-12.696,-72.802,170.594,31.537,155.936
C08398=1051.801,-12.447,-72.816,170.596,31.538,155.936
C08399=1051.809,-12.197,-72.830,170.598,31.540,155.936
C08400=1051.814,-11.948,-72.844,170.599,31.542,155.937
C08401=1051.820,-11.698,-72.859,170.601,31.544,155.937
C08402=1051.827,-11.449,-72.872,170.603,31.546,155.937
C08403=1051.833,-11.199,-72.887,170.604,31.548,155.938
C08404=1051.838,-10.950,-72.901,170.606,31.549,155.938
C08405=1051.846,-10.700,-72.915,170.608,31.551,155.938
C08406=1051.851,-10.451,-72.929,170.610,31.553,155.938
C08407=1051.857,-10.201,-72.944,170.611,31.555,155.938
C08408=1051.865,-9.952,-72.959,170.613,31.557,155.939
C08409=1051.870,-9.702,-72.972,170.615,31.559,155.939
C08410=1051.876,-9.453,-72.987,170.617,31.561,155.939
C08411=1051.882,-9.203,-73.001,170.619,31.563,155.940
C08412=1051.889,-8.954,-73.016,170.620,31.564,155.940
C08413=1051.895,-8.705,-73.030,170.621,31.566,155.940
C08414=1051.901,-8.454,-73.044,170.623,31.568,155.940
C08415=1051.908,-8.205,-73.059,170.625,31.570,155.940
C08416=1051.913,-7.955,-73.073,170.627,31.572,155.941
C08417=1051.920,-7.706,-73.088,170.629,31.574,155.941
C08418=1051.926,-7.457,-73.101,170.631,31.576,155.941
C08419=1051.932,-7.207,-73.116,170.632,31.578,155.942
C08420=1051.939,-6.957,-73.131,170.634,31.579,155.942
C08421=1051.945,-6.708,-73.145,170.636,31.581,155.942
C08422=1051.951,-6.458,-73.159,170.637,31.583,155.942
C08423=1051.957,-6.209,-73.173,170.639,31.585,155.942
C08424=1051.964,-5.960,-73.188,170.641,31.587,155.943
C08425=1051.970,-5.709,-73.203,170.642,31.589,155.943
C08426=1051.976,-5.461,-73.217,170.644,31.590,155.943
C08427=1051.983,-5.211,-73.232,170.646,31.592,155.943
C08428=1051.989,-4.961,-73.247,170.648,31.595,155.944
C08429=1051.995,-4.712,-73.260,170.650,31.596,155.944
C08430=1052.002,-4.463,-73.275,170.652,31.598,155.944
C08431=1052.008,-4.213,-73.290,170.652,31.600,155.945
C08432=1052.014,-3.964,-73.304,170.654,31.602,155.945
C08433=1052.021,-3.714,-73.318,170.656,31.604,155.945
C08434=1052.027,-3.464,-73.333,170.658,31.606,155.945
C08435=1052.033,-3.215,-73.347,170.660,31.607,155.945
C08436=1052.040,-2.932,-73.364,170.662,31.610,155.946
C08437=1052.047,-2.650,-73.380,170.664,31.612,155.946
C08438=1052.054,-2.367,-73.398,170.666,31.614,155.946
C08439=1052.061,-2.085,-73.414,170.668,31.616,155.947
C08440=1052.067,-1.835,-73.429,170.669,31.618,155.947
C08441=1052.073,-1.586,-73.444,170.671,31.621,155.947
C08442=1052.079,-1.336,-73.458,170.672,31.622,155.948
C08443=1052.085,-1.087,-73.473,170.674,31.625,155.948
C08444=1052.091,-0.837,-73.488,170.676,31.626,155.948
C08445=1052.098,-0.588,-73.502,170.678,31.628,155.948
C08446=1052.103,-0.338,-73.518,170.680,31.630,155.949
C08447=1052.109,-0.089,-73.533,170.681,31.632,155.949
C08448=1052.115,0.161,-73.548,170.683,31.634,155.949
C08449=1052.121,0.410,-73.562,170.685,31.636,155.950
C08450=1052.127,0.660,-73.577,170.686,31.639,155.950
C08451=1052.134,0.909,-73.592,170.687,31.640,155.950
C08452=1052.140,1.159,-73.607,170.689,31.642,155.950
C08453=1052.146,1.408,-73.622,170.691,31.644,155.951
C08454=1052.152,1.658,-73.636,170.693,31.646,155.951
C08455=1052.159,1.907,-73.651,170.695,31.648,155.951
C08456=1052.165,2.156,-73.666,170.696,31.650,155.951
C08457=1052.171,2.406,-73.681,170.698,31.652,155.952
C08458=1052.177,2.655,-73.696,170.700,31.654,155.952
C08459=1052.184,2.905,-73.711,170.701,31.656,155.952
C08460=1052.190,3.154,-73.725,170.703,31.658,155.953
C08461=1052.196,3.404,-73.740,170.704,31.660,155.953
C08462=1052.202,3.653,-73.755,170.706,31.662,155.953
C08463=1052.207,3.903,-73.770,170.708,31.664,155.953
C08464=1052.214,4.152,-73.785,170.710,31.666,155.954
C08465=1052.220,4.402,-73.800,170.712,31.668,155.954
C08466=1052.226,4.652,-73.815,170.713,31.670,155.954
C08467=1052.233,4.901,-73.830,170.715,31.672,155.954
C08468=1052.239,5.150,-73.845,170.717,31.674,155.955
C08469=1052.245,5.400,-73.860,170.718,31.676,155.955
C08470=1052.251,5.650,-73.875,170.719,31.677,155.955
C08471=1052.258,5.899,-73.890,170.721,31.680,155.956
C08472=1052.264,6.148,-73.904,170.723,31.682,155.956
C08473=1052.270,6.398,-73.919,170.725,31.684,155.956
C08474=1052.276,6.647,-73.935,170.727,31.686,155.956
C08475=1052.282,6.897,-73.950,170.728,31.688,155.957
C08476=1052.289,7.146,-73.965,170.730,31.690,155.957
C08477=1052.294,7.395,-73.980,170.732,31.691,155.957
C08478=1052.301,7.645,-73.995,170.734,31.693,155.957
C08479=1052.307,7.895,-74.010,170.734,31.695,155.958
C08480=1052.314,8.144,-74.026,170.736,31.697,155.958
C08481=1052.320,8.393,-74.040,170.738,31.700,155.958
C08482=1052.327,8.643,-74.055,170.740,31.702,155.959
C08483=1052.332,8.892,-74.071,170.742,31.704,155.959
C08484=1052.338,9.142,-74.086,170.743,31.705,155.959
C08485=1052.344,9.392,-74.100,170.745,31.707,155.959
C08486=1052.351,9.641,-74.116,170.747,31.709,155.960
C08487=1052.358,9.890,-74.131,170.749,31.711,155.960
C08488=1052.364,10.140,-74.146,170.750,31.713,155.960
C08489=1052.370,10.390,-74.161,170.751,31.715,155.961
C08490=1052.377,10.639,-74.177,170.753,31.718,155.961
C08491=1052.382,10.888,-74.192,170.755,31.719,155.961
C08492=1052.388,11.138,-74.207,170.757,31.721,155.961
C08493=1052.395,11.387,-74.222,170.758,31.723,155.962
C08494=1052.402,11.636,-74.237,170.760,31.725,155.962
C08495=1052.408,11.886,-74.252,170.762,31.727,155.962
C08496=1052.414,12.136,-74.267,170.764,31.729,155.963
C08497=1052.421,12.385,-74.283,170.765,31.731,155.963
C08498=1052.427,12.635,-74.298,170.767,31.733,155.963
C08499=1052.433,12.884,-74.313,170.768,31.735,155.963
C08500=1052.440,13.169,-74.331,170.770,31.737,155.964
C08501=1052.448,13.453,-74.347,170.772,31.740,155.964
C08502=1052.455,13.737,-74.365,170.774,31.742,155.964
C08503=1052.462,14.022,-74.383,170.776,31.744,155.965
C08504=1052.468,14.271,-74.398,170.778,31.746,155.965
C08505=1052.474,14.520,-74.414,170.779,31.748,155.965
C08506=1052.481,14.770,-74.429,170.781,31.750,155.965
C08507=1052.486,15.020,-74.444,170.783,31.752,155.966
C08508=1052.493,15.269,-74.460,170.784,31.754,155.966
C08509=1052.499,15.519,-74.475,170.785,31.756,155.966
C08510=1052.505,15.768,-74.491,170.787,31.758,155.967
C08511=1052.512,16.018,-74.506,170.789,31.760,155.967
C08512=1052.518,16.267,-74.521,170.791,31.762,155.967
C08513=1052.524,16.517,-74.537,170.792,31.764,155.968
C08514=1052.530,16.766,-74.552,170.794,31.766,155.968
C08515=1052.536,17.016,-74.569,170.796,31.769,155.968
C08516=1052.543,17.265,-74.584,170.798,31.771,155.968
C08517=1052.549,17.514,-74.599,170.799,31.773,155.969
C08518=1052.554,17.764,-74.614,170.801,31.775,155.969
C08519=1052.561,18.013,-74.630,170.802,31.777,155.969
C08520=1052.567,18.263,-74.646,170.804,31.779,155.970
C08521=1052.573,18.512,-74.661,170.805,31.781,155.970
C08522=1052.580,18.761,-74.676,170.807,31.783,155.970
C08523=1052.586,19.011,-74.693,170.809,31.785,155.970
C08524=1052.592,19.260,-74.707,170.811,31.787,155.971
C08525=1052.598,19.510,-74.724,170.812,31.789,155.971
C08526=1052.605,19.759,-74.739,170.814,31.791,155.971
C08527=1052.610,20.009,-74.755,170.816,31.793,155.972
C08528=1052.617,20.258,-74.771,170.817,31.795,155.972
C08529=1052.623,20.508,-74.786,170.818,31.797,155.972
C08530=1052.629,20.757,-74.802,170.820,31.799,155.973
C08531=1052.635,21.007,-74.817,170.822,31.801,155.973
C08532=1052.642,21.256,-74.833,170.823,31.803,155.973
C08533=1052.648,21.505,-74.849,170.825,31.805,155.973
C08534=1052.654,21.755,-74.864,170.827,31.808,155.974
C08535=1052.660,22.004,-74.880,170.829,31.810,155.974
C08536=1052.667,22.253,-74.896,170.830,31.812,155.974
C08537=1052.672,22.503,-74.912,170.832,31.814,155.975
C08538=1052.679,22.752,-74.927,170.834,31.816,155.975
C08539=1052.685,23.002,-74.944,170.834,31.818,155.975
C08540=1052.691,23.252,-74.959,170.836,31.820,155.976
C08541=1052.697,23.501,-74.975,170.838,31.822,155.976
C08542=1052.703,23.750,-74.991,170.840,31.825,155.976
C08543=1052.710,24.000,-75.006,170.841,31.827,155.977
C08544=1052.716,24.249,-75.022,170.843,31.829,155.977
C08545=1052.722,24.498,-75.038,170.845,31.831,155.977
C08546=1052.728,24.748,-75.053,170.847,31.833,155.977
C08547=1052.734,24.997,-75.070,170.848,31.835,155.978
C08548=1052.741,25.246,-75.085,170.850,31.837,155.978
C08549=1052.747,25.496,-75.102,170.852,31.839,155.978
C08550=1052.754,25.746,-75.117,170.852,31.841,155.979
C08551=1052.759,25.995,-75.133,170.854,31.843,155.979
C08552=1052.766,26.244,-75.149,170.856,31.845,155.979
C08553=1052.772,26.494,-75.165,170.858,31.847,155.980
C08554=1052.778,26.744,-75.181,170.859,31.849,155.980
C08555=1052.784,26.993,-75.196,170.861,31.851,155.980
C08556=1052.790,27.242,-75.213,170.863,31.853,155.980
C08557=1052.797,27.491,-75.228,170.864,31.855,155.981
C08558=1052.803,27.741,-75.244,170.866,31.857,155.981
C08559=1052.809,27.990,-75.261,170.868,31.859,155.981
C08560=1052.815,28.240,-75.276,170.869,31.862,155.982
C08561=1052.822,28.490,-75.292,170.870,31.864,155.982
C08562=1052.828,28.739,-75.309,170.872,31.866,155.982
C08563=1052.834,28.988,-75.325,170.874,31.868,155.983
C08564=1052.841,29.274,-75.343,170.876,31.870,155.983
C08565=1052.848,29.560,-75.362,170.878,31.873,155.983
C08566=1052.855,29.846,-75.380,170.880,31.876,155.984
C08567=1052.862,30.131,-75.398,170.881,31.878,155.984
C08568=1052.868,30.380,-75.414,170.883,31.880,155.984
C08569=1052.875,30.630,-75.431,170.885,31.882,155.985
C08570=1052.881,30.880,-75.447,170.887,31.884,155.985
C08571=1052.887,31.129,-75.463,170.887,31.886,155.985
C08572=1052.893,31.378,-75.479,170.889,31.888,155.986
C08573=1052.899,31.627,-75.495,170.891,31.891,155.986
C08574=1052.905,31.877,-75.511,170.892,31.892,155.986
C08575=1052.911,32.126,-75.528,170.894,31.895,155.987
C08576=1052.917,32.375,-75.544,170.896,31.897,155.987
C08577=1052.924,32.625,-75.560,170.897,31.899,155.987
C08578=1052.930,32.874,-75.576,170.899,31.901,155.988
C08579=1052.936,33.124,-75.592,170.901,31.903,155.988
C08580=1052.942,33.373,-75.609,170.903,31.905,155.988
C08581=1052.948,33.622,-75.625,170.904,31.907,155.988
C08582=1052.954,33.872,-75.641,170.905,31.909,155.989
C08583=1052.962,34.122,-75.657,170.907,31.912,155.989
C08584=1052.968,34.371,-75.673,170.908,31.914,155.990
C08585=1052.973,34.620,-75.690,170.910,31.916,155.990
C08586=1052.979,34.870,-75.706,170.912,31.918,155.990
C08587=1052.985,35.119,-75.722,170.913,31.920,155.990
C08588=1052.991,35.368,-75.738,170.915,31.922,155.991
C08589=1052.999,35.618,-75.754,170.917,31.924,155.991
C08590=1053.005,35.867,-75.771,170.919,31.926,155.991
C08591=1053.011,36.117,-75.787,170.920,31.929,155.992
C08592=1053.016,36.366,-75.803,170.922,31.931,155.992
C08593=1053.023,36.616,-75.820,170.923,31.933,155.992
C08594=1053.029,36.865,-75.836,170.924,31.935,155.993
C08595=1053.036,37.114,-75.852,170.926,31.937,155.993
C08596=1053.042,37.363,-75.869,170.928,31.939,155.993
C08597=1053.048,37.613,-75.885,170.929,31.941,155.994
C08598=1053.054,37.863,-75.902,170.931,31.944,155.994
C08599=1053.060,38.112,-75.918,170.933,31.946,155.994
C08600=1053.066,38.361,-75.934,170.934,31.948,155.995
C08601=1053.073,38.610,-75.951,170.936,31.950,155.995
C08602=1053.079,38.860,-75.968,170.938,31.953,155.995
C08603=1053.085,39.109,-75.984,170.939,31.955,155.996
C08604=1053.091,39.359,-76.000,170.940,31.957,155.996
C08605=1053.097,39.608,-76.016,170.942,31.959,155.996
C08606=1053.103,39.857,-76.033,170.944,31.961,155.996
C08607=1053.110,40.107,-76.050,170.945,31.963,155.997
C08608=1053.116,40.356,-76.066,170.947,31.965,155.997
C08609=1053.122,40.606,-76.083,170.949,31.967,155.997
C08610=1053.127,40.855,-76.100,170.950,31.969,155.998
C08611=1053.134,41.105,-76.117,170.952,31.972,155.998
C08612=1053.140,41.354,-76.133,170.954,31.974,155.998
C08613=1053.146,41.603,-76.149,170.955,31.976,155.999
C08614=1053.152,41.852,-76.166,170.957,31.978,155.999
C08615=1053.158,42.102,-76.183,170.959,31.980,155.999
C08616=1053.164,42.352,-76.199,170.959,31.983,156.000
C08617=1053.171,42.600,-76.216,170.961,31.985,156.000
C08618=1053.177,42.850,-76.232,170.963,31.987,156.000
C08619=1053.183,43.100,-76.249,170.964,31.989,156.001
C08620=1053.189,43.348,-76.266,170.966,31.992,156.001
C08621=1053.195,43.598,-76.282,170.968,31.994,156.001
C08622=1053.201,43.848,-76.299,170.969,31.996,156.002
C08623=1053.207,44.097,-76.316,170.971,31.998,156.002
C08624=1053.213,44.346,-76.333,170.973,32.000,156.002
C08625=1053.220,44.595,-76.350,170.974,32.002,156.003
C08626=1053.226,44.845,-76.367,170.976,32.005,156.003
C08627=1053.231,45.095,-76.383,170.977,32.007,156.003
C08628=1053.238,45.380,-76.403,170.979,32.010,156.004
C08629=1053.246,45.665,-76.422,170.980,32.012,156.004
C08630=1053.252,45.952,-76.441,170.982,32.014,156.005
C08631=1053.259,46.237,-76.460,170.984,32.017,156.005
C08632=1053.265,46.487,-76.477,170.986,32.020,156.005
C08633=1053.271,46.736,-76.494,170.988,32.022,156.006
C08634=1053.277,46.985,-76.511,170.989,32.024,156.006
C08635=1053.283,47.235,-76.529,170.991,32.026,156.006
C08636=1053.289,47.484,-76.545,170.993,32.028,156.007
C08637=1053.296,47.733,-76.562,170.994,32.030,156.007
C08638=1053.301,47.983,-76.579,170.996,32.033,156.007
C08639=1053.308,48.232,-76.596,170.997,32.035,156.008
C08640=1053.314,48.482,-76.612,170.998,32.037,156.008
C08641=1053.319,48.731,-76.630,171.000,32.039,156.008
C08642=1053.326,48.981,-76.646,171.002,32.042,156.009
C08643=1053.332,49.229,-76.663,171.003,32.044,156.009
C08644=1053.337,49.479,-76.680,171.005,32.046,156.009
C08645=1053.344,49.729,-76.698,171.007,32.048,156.010
C08646=1053.350,49.977,-76.715,171.008,32.050,156.010
C08647=1053.356,50.227,-76.731,171.010,32.052,156.010
C08648=1053.362,50.476,-76.749,171.012,32.055,156.011
C08649=1053.368,50.726,-76.765,171.013,32.057,156.011
C08650=1053.374,50.975,-76.783,171.015,32.059,156.011
C08651=1053.381,51.224,-76.800,171.016,32.062,156.012
C08652=1053.387,51.474,-76.816,171.017,32.064,156.012
C08653=1053.393,51.723,-76.834,171.019,32.066,156.013
C08654=1053.399,51.973,-76.850,171.021,32.068,156.013
C08655=1053.405,52.221,-76.867,171.022,32.070,156.013
C08656=1053.411,52.471,-76.885,171.024,32.072,156.014
C08657=1053.417,52.720,-76.902,171.025,32.074,156.014
C08658=1053.424,52.970,-76.919,171.027,32.077,156.014
C08659=1053.429,53.219,-76.936,171.029,32.079,156.015
C08660=1053.436,53.469,-76.953,171.030,32.081,156.015
C08661=1053.442,53.718,-76.970,171.032,32.084,156.015
C08662=1053.448,53.967,-76.988,171.034,32.086,156.016
C08663=1053.454,54.217,-77.004,171.035,32.088,156.016
C08664=1053.460,54.466,-77.022,171.036,32.090,156.016
C08665=1053.467,54.715,-77.039,171.038,32.092,156.017
C08666=1053.473,54.964,-77.056,171.039,32.094,156.017
C08667=1053.479,55.214,-77.073,171.041,32.096,156.017
C08668=1053.485,55.463,-77.090,171.043,32.099,156.018
C08669=1053.492,55.712,-77.108,171.044,32.101,156.018
C08670=1053.497,55.962,-77.125,171.046,32.103,156.018
C08671=1053.503,56.211,-77.142,171.048,32.106,156.019
C08672=1053.509,56.461,-77.159,171.049,32.108,156.019
C08673=1053.516,56.709,-77.176,171.051,32.110,156.019
C08674=1053.523,56.959,-77.194,171.053,32.112,156.020
C08675=1053.528,57.208,-77.211,171.054,32.114,156.020
C08676=1053.535,57.458,-77.228,171.056,32.116,156.020
C08677=1053.540,57.707,-77.246,171.057,32.118,156.021
C08678=1053.547,57.956,-77.263,171.058,32.121,156.021
C08679=1053.553,58.205,-77.280,171.060,32.123,156.021
C08680=1053.559,58.455,-77.297,171.062,32.125,156.022
C08681=1053.565,58.704,-77.314,171.063,32.127,156.022
C08682=1053.571,58.954,-77.332,171.065,32.130,156.022
C08683=1053.578,59.203,-77.349,171.067,32.132,156.023
C08684=1053.585,59.452,-77.366,171.068,32.134,156.023
C08685=1053.591,59.702,-77.384,171.070,32.136,156.023
C08686=1053.597,59.951,-77.401,171.072,32.138,156.024
C08687=1053.603,60.201,-77.418,171.073,32.140,156.024
C08688=1053.609,60.450,-77.435,171.075,32.142,156.024
C08689=1053.615,60.699,-77.453,171.077,32.145,156.025
C08690=1053.621,60.948,-77.470,171.077,32.147,156.025
C08691=1053.628,61.198,-77.488,171.079,32.149,156.025
C08692=1053.635,61.483,-77.508,171.081,32.152,156.026
C08693=1053.642,61.768,-77.528,171.083,32.154,156.026
C08694=1053.650,62.054,-77.547,171.085,32.156,156.026
C08695=1053.657,62.340,-77.567,171.087,32.159,156.027
C08696=1053.663,62.589,-77.585,171.088,32.161,156.027
C08697=1053.669,62.838,-77.602,171.090,32.163,156.028
C08698=1053.676,63.087,-77.619,171.092,32.166,156.028
C08699=1053.681,63.337,-77.637,171.093,32.168,156.028
C08700=1053.688,63.586,-77.654,171.095,32.170,156.029
C08701=1053.694,63.836,-77.672,171.097,32.172,156.029
C08702=1053.701,64.084,-77.689,171.098,32.174,156.029
C08703=1053.707,64.334,-77.707,171.099,32.176,156.030
C08704=1053.713,64.583,-77.724,171.101,32.178,156.030
C08705=1053.719,64.833,-77.742,171.102,32.181,156.030
C08706=1053.725,65.082,-77.760,171.104,32.183,156.031
C08707=1053.731,65.331,-77.778,171.106,32.185,156.031
C08708=1053.738,65.581,-77.795,171.107,32.188,156.031
C08709=1053.743,65.830,-77.812,171.109,32.190,156.032
C08710=1053.750,66.079,-77.831,171.111,32.192,156.032
C08711=1053.756,66.328,-77.848,171.112,32.194,156.032
C08712=1053.762,66.577,-77.866,171.114,32.196,156.033
C08713=1053.768,66.827,-77.884,171.116,32.199,156.033
C08714=1053.774,67.076,-77.901,171.117,32.201,156.033
C08715=1053.780,67.326,-77.919,171.119,32.203,156.034
C08716=1053.787,67.575,-77.937,171.121,32.206,156.034
C08717=1053.792,67.824,-77.954,171.121,32.208,156.034
C08718=1053.799,68.073,-77.972,171.123,32.210,156.035
C08719=1053.805,68.322,-77.990,171.125,32.212,156.035
C08720=1053.811,68.572,-78.008,171.126,32.214,156.035
C08721=1053.817,68.822,-78.026,171.128,32.217,156.036
C08722=1053.823,69.071,-78.043,171.130,32.219,156.036
C08723=1053.829,69.320,-78.061,171.131,32.221,156.037
C08724=1053.836,69.569,-78.079,171.133,32.224,156.037
C08725=1053.841,69.818,-78.097,171.135,32.226,156.037
C08726=1053.848,70.068,-78.114,171.136,32.227,156.038
C08727=1053.854,70.317,-78.132,171.138,32.230,156.038
C08728=1053.860,70.566,-78.150,171.140,32.232,156.038
C08729=1053.866,70.816,-78.168,171.141,32.235,156.039
C08730=1053.872,71.065,-78.186,171.143,32.237,156.039
C08731=1053.878,71.315,-78.204,171.145,32.239,156.039
C08732=1053.884,71.564,-78.223,171.145,32.241,156.040
C08733=1053.890,71.813,-78.240,171.147,32.243,156.040
C08734=1053.897,72.062,-78.257,171.148,32.246,156.040
C08735=1053.903,72.311,-78.276,171.150,32.248,156.041
C08736=1053.909,72.560,-78.294,171.152,32.251,156.041
C08737=1053.915,72.810,-78.312,171.153,32.253,156.042
C08738=1053.921,73.059,-78.330,171.155,32.255,156.042
C08739=1053.927,73.308,-78.348,171.157,32.257,156.042
C08740=1053.933,73.558,-78.366,171.158,32.259,156.043
C08741=1053.939,73.807,-78.384,171.160,32.262,156.043
C08742=1053.945,74.056,-78.402,171.162,32.264,156.043
C08743=1053.951,74.306,-78.420,171.163,32.266,156.044
C08744=1053.957,74.555,-78.439,171.165,32.268,156.044
C08745=1053.964,74.804,-78.456,171.167,32.271,156.044
C08746=1053.970,75.053,-78.473,171.168,32.273,156.045
C08747=1053.976,75.303,-78.492,171.169,32.275,156.045
C08748=1053.982,75.552,-78.510,171.171,32.278,156.045
C08749=1053.988,75.801,-78.528,171.172,32.280,156.046
C08750=1053.994,76.050,-78.546,171.174,32.282,156.046
C08751=1054.000,76.300,-78.564,171.176,32.284,156.047
C08752=1054.006,76.549,-78.582,171.177,32.286,156.047
C08753=1054.012,76.798,-78.600,171.179,32.289,156.047
C08754=1054.019,77.047,-78.619,171.181,32.291,156.048
C08755=1054.025,77.297,-78.637,171.182,32.293,156.048
C08756=1054.032,77.583,-78.658,171.184,32.296,156.048
C08757=1054.039,77.867,-78.678,171.186,32.298,156.049
C08758=1054.045,78.153,-78.699,171.188,32.301,156.049
C08759=1054.052,78.438,-78.720,171.190,32.303,156.050
C08760=1054.058,78.681,-78.738,171.191,32.305,156.050
C08761=1054.065,78.925,-78.756,171.193,32.308,156.050
C08762=1054.071,79.168,-78.774,171.194,32.310,156.051
C08763=1054.076,79.411,-78.791,171.195,32.313,156.051
C08764=1054.082,79.654,-78.809,171.197,32.315,156.051
C08765=1054.088,79.897,-78.827,171.199,32.317,156.052
C08766=1054.093,80.140,-78.845,171.200,32.319,156.052
C08767=1054.099,80.383,-78.863,171.202,32.321,156.052
C08768=1054.105,80.633,-78.882,171.203,32.324,156.053
C08769=1054.112,80.882,-78.900,171.205,32.326,156.053
C08770=1054.118,81.131,-78.918,171.207,32.328,156.054
C08771=1054.124,81.380,-78.937,171.208,32.330,156.054
C08772=1054.130,81.629,-78.955,171.210,32.333,156.054
C08773=1054.136,81.879,-78.974,171.212,32.335,156.055
C08774=1054.142,82.128,-78.992,171.213,32.338,156.055
C08775=1054.148,82.377,-79.010,171.215,32.340,156.055
C08776=1054.154,82.626,-79.029,171.217,32.342,156.056
C08777=1054.160,82.875,-79.047,171.218,32.344,156.056
C08778=1054.166,83.126,-79.066,171.219,32.347,156.056
C08779=1054.172,83.375,-79.084,171.221,32.349,156.057
C08780=1054.178,83.623,-79.103,171.222,32.351,156.057
C08781=1054.184,83.873,-79.121,171.224,32.353,156.058
C08782=1054.191,84.122,-79.139,171.226,32.356,156.058
C08783=1054.196,84.371,-79.159,171.227,32.358,156.058
C08784=1054.203,84.620,-79.177,171.229,32.361,156.059
C08785=1054.208,84.869,-79.195,171.231,32.363,156.059
C08786=1054.215,85.119,-79.213,171.232,32.365,156.059
C08787=1054.221,85.368,-79.232,171.234,32.367,156.060
C08788=1054.227,85.617,-79.251,171.236,32.369,156.060
C08789=1054.233,85.867,-79.269,171.237,32.372,156.060
C08790=1054.239,86.116,-79.288,171.239,32.374,156.061
C08791=1054.246,86.365,-79.307,171.241,32.377,156.061
C08792=1054.251,86.614,-79.325,171.242,32.378,156.061
C08793=1054.257,86.864,-79.343,171.244,32.381,156.062
C08794=1054.263,87.113,-79.362,171.246,32.383,156.062
C08795=1054.270,87.362,-79.381,171.246,32.386,156.063
C08796=1054.275,87.611,-79.400,171.248,32.388,156.063
C08797=1054.282,87.860,-79.419,171.250,32.390,156.063
C08798=1054.288,88.110,-79.436,171.251,32.392,156.064
C08799=1054.294,88.359,-79.455,171.253,32.394,156.064
C08800=1054.300,88.608,-79.473,171.255,32.397,156.064
C08801=1054.306,88.857,-79.493,171.256,32.399,156.065
C08802=1054.312,89.106,-79.511,171.258,32.401,156.065
C08803=1054.319,89.355,-79.530,171.260,32.403,156.065
C08804=1054.325,89.605,-79.549,171.261,32.406,156.066
C08805=1054.331,89.855,-79.567,171.263,32.408,156.066
C08806=1054.337,90.104,-79.586,171.265,32.410,156.067
C08807=1054.343,90.353,-79.604,171.266,32.413,156.067
C08808=1054.349,90.602,-79.624,171.268,32.415,156.067
C08809=1054.356,90.851,-79.642,171.270,32.417,156.068
C08810=1054.361,91.101,-79.662,171.271,32.419,156.068
C08811=1054.368,91.350,-79.680,171.273,32.422,156.068
C08812=1054.373,91.599,-79.699,171.275,32.424,156.069
C08813=1054.379,91.848,-79.718,171.275,32.426,156.069
C08814=1054.386,92.097,-79.736,171.277,32.429,156.070
C08815=1054.391,92.346,-79.756,171.279,32.431,156.070
C08816=1054.398,92.595,-79.774,171.280,32.434,156.070
C08817=1054.403,92.845,-79.793,171.282,32.436,156.071
C08818=1054.410,93.094,-79.812,171.284,32.438,156.071
C08819=1054.416,93.343,-79.831,171.285,32.440,156.071
C08820=1054.423,93.640,-79.854,171.287,32.443,156.072
C08821=1054.429,93.938,-79.876,171.289,32.446,156.072
C08822=1054.437,94.236,-79.899,171.291,32.449,156.073
C08823=1054.444,94.533,-79.922,171.293,32.451,156.073
C08824=1054.450,94.782,-79.941,171.295,32.454,156.074
C08825=1054.456,95.032,-79.960,171.297,32.456,156.074
C08826=1054.462,95.281,-79.979,171.298,32.458,156.074
C08827=1054.469,95.530,-79.997,171.300,32.460,156.075
C08828=1054.474,95.780,-80.017,171.302,32.463,156.075
C08829=1054.481,96.029,-80.035,171.303,32.465,156.075
C08830=1054.486,96.278,-80.055,171.305,32.468,156.076
C08831=1054.492,96.528,-80.074,171.306,32.470,156.076
C08832=1054.499,96.776,-80.093,171.307,32.472,156.077
C08833=1054.504,97.025,-80.112,171.309,32.474,156.077
C08834=1054.511,97.275,-80.131,171.311,32.477,156.077
C08835=1054.517,97.524,-80.150,171.313,32.479,156.078
C08836=1054.523,97.773,-80.169,171.314,32.481,156.078
C08837=1054.529,98.023,-80.188,171.316,32.483,156.078
C08838=1054.535,98.271,-80.208,171.318,32.486,156.079
C08839=1054.541,98.520,-80.227,171.319,32.488,156.079
C08840=1054.548,98.770,-80.245,171.321,32.491,156.080
C08841=1054.553,99.019,-80.265,171.323,32.493,156.080
C08842=1054.560,99.268,-80.283,171.324,32.495,156.080
C08843=1054.566,99.517,-80.303,171.326,32.497,156.081
C08844=1054.571,99.766,-80.323,171.328,32.500,156.081
C08845=1054.578,100.016,-80.341,171.329,32.502,156.081
C08846=1054.583,100.265,-80.360,171.331,32.504,156.082
C08847=1054.590,100.514,-80.379,171.333,32.506,156.082
C08848=1054.596,100.763,-80.399,171.335,32.509,156.082
C08849=1054.602,101.012,-80.418,171.336,32.511,156.083
C08850=1054.608,101.261,-80.437,171.338,32.514,156.083
C08851=1054.614,101.510,-80.457,171.340,32.516,156.084
C08852=1054.620,101.760,-80.476,171.340,32.518,156.084
C08853=1054.626,102.010,-80.496,171.342,32.521,156.084
C08854=1054.633,102.258,-80.515,171.344,32.523,156.085
C08855=1054.638,102.508,-80.534,171.345,32.525,156.085
C08856=1054.644,102.757,-80.554,171.347,32.528,156.086
C08857=1054.650,103.006,-80.574,171.349,32.530,156.086
C08858=1054.656,103.255,-80.593,171.350,32.532,156.086
C08859=1054.662,103.505,-80.611,171.352,32.535,156.087
C08860=1054.668,103.753,-80.631,171.354,32.537,156.087
C08861=1054.674,104.003,-80.651,171.355,32.540,156.087
C08862=1054.680,104.252,-80.670,171.357,32.542,156.088
C08863=1054.686,104.501,-80.690,171.359,32.544,156.088
C08864=1054.692,104.750,-80.708,171.361,32.546,156.088
C08865=1054.698,104.999,-80.728,171.362,32.549,156.089
C08866=1054.704,105.248,-80.748,171.364,32.551,156.089
C08867=1054.710,105.497,-80.768,171.366,32.553,156.090
C08868=1054.715,105.747,-80.787,171.367,32.556,156.090
C08869=1054.722,105.997,-80.807,171.369,32.558,156.090
C08870=1054.728,106.245,-80.826,171.371,32.561,156.091
C08871=1054.734,106.495,-80.845,171.372,32.562,156.091
C08872=1054.740,106.744,-80.865,171.374,32.565,156.092
C08873=1054.746,106.993,-80.884,171.375,32.568,156.092
C08874=1054.752,107.242,-80.904,171.377,32.570,156.092
C08875=1054.758,107.491,-80.923,171.378,32.572,156.093
C08876=1054.764,107.740,-80.943,171.380,32.574,156.093
C08877=1054.770,107.990,-80.962,171.382,32.577,156.093
C08878=1054.776,108.239,-80.982,171.383,32.579,156.094
C08879=1054.782,108.488,-81.002,171.385,32.581,156.094
C08880=1054.788,108.737,-81.022,171.387,32.584,156.095
C08881=1054.794,108.986,-81.042,171.389,32.586,156.095
C08882=1054.801,109.235,-81.060,171.390,32.589,156.095
C08883=1054.807,109.484,-81.080,171.392,32.591,156.096
C08884=1054.813,109.770,-81.103,171.394,32.593,156.096
C08885=1054.820,110.055,-81.125,171.396,32.596,156.097
C08886=1054.827,110.340,-81.147,171.398,32.598,156.097
C08887=1054.835,110.625,-81.170,171.400,32.601,156.097
C08888=1054.841,110.875,-81.190,171.402,32.604,156.098
C08889=1054.847,111.124,-81.210,171.403,32.606,156.098
C08890=1054.853,111.373,-81.229,171.405,32.608,156.099
C08891=1054.859,111.622,-81.249,171.407,32.611,156.099
C08892=1054.865,111.871,-81.269,171.408,32.613,156.099
C08893=1054.870,112.120,-81.288,171.410,32.615,156.100
C08894=1054.877,112.370,-81.308,171.412,32.618,156.100
C08895=1054.883,112.619,-81.328,171.414,32.620,156.100
C08896=1054.889,112.868,-81.348,171.415,32.622,156.101
C08897=1054.895,113.117,-81.368,171.416,32.624,156.101
C08898=1054.901,113.366,-81.388,171.418,32.627,156.102
C08899=1054.907,113.615,-81.408,171.419,32.630,156.102
C08900=1054.913,113.865,-81.427,171.421,32.632,156.102
C08901=1054.919,114.113,-81.447,171.423,32.634,156.103
C08902=1054.924,114.362,-81.468,171.425,32.637,156.103
C08903=1054.930,114.611,-81.488,171.426,32.639,156.104
C08904=1054.936,114.861,-81.507,171.428,32.641,156.104
C08905=1054.942,115.110,-81.527,171.430,32.644,156.104
C08906=1054.948,115.359,-81.547,171.431,32.646,156.105
C08907=1054.954,115.608,-81.568,171.433,32.649,156.105
C08908=1054.960,115.857,-81.588,171.435,32.651,156.106
C08909=1054.965,116.106,-81.607,171.437,32.654,156.106
C08910=1054.972,116.356,-81.627,171.438,32.656,156.106
C08911=1054.977,116.605,-81.648,171.440,32.658,156.107
C08912=1054.983,116.854,-81.668,171.442,32.661,156.107
C08913=1054.989,117.103,-81.688,171.444,32.663,156.108
C08914=1054.995,117.351,-81.708,171.445,32.665,156.108
C08915=1055.001,117.601,-81.729,171.447,32.668,156.108
C08916=1055.007,117.850,-81.749,171.449,32.671,156.109
C08917=1055.013,118.100,-81.768,171.450,32.673,156.109
C08918=1055.019,118.348,-81.788,171.452,32.675,156.110
C08919=1055.025,118.598,-81.809,171.454,32.678,156.110
C08920=1055.031,118.847,-81.829,171.456,32.680,156.110
C08921=1055.036,119.096,-81.849,171.457,32.682,156.111
C08922=1055.042,119.345,-81.869,171.459,32.685,156.111
C08923=1055.048,119.594,-81.889,171.461,32.687,156.111
C08924=1055.054,119.843,-81.909,171.462,32.689,156.112
C08925=1055.060,120.092,-81.929,171.463,32.692,156.112
C08926=1055.066,120.341,-81.950,171.465,32.694,156.113
C08927=1055.072,120.591,-81.970,171.467,32.697,156.113
C08928=1055.078,120.840,-81.990,171.469,32.699,156.114
C08929=1055.084,121.088,-82.010,171.470,32.701,156.114
C08930=1055.090,121.338,-82.031,171.472,32.704,156.114
C08931=1055.096,121.587,-82.051,171.474,32.706,156.115
C08932=1055.102,121.836,-82.071,171.476,32.708,156.115
C08933=1055.108,122.086,-82.092,171.477,32.711,156.115
C08934=1055.114,122.334,-82.112,171.479,32.713,156.116
C08935=1055.120,122.583,-82.132,171.481,32.716,156.116
C08936=1055.126,122.833,-82.153,171.483,32.718,156.117
C08937=1055.132,123.082,-82.173,171.484,32.721,156.117
C08938=1055.138,123.331,-82.193,171.486,32.723,156.117
C08939=1055.144,123.580,-82.213,171.488,32.725,156.118
C08940=1055.150,123.829,-82.234,171.490,32.728,156.118
C08941=1055.156,124.078,-82.254,171.491,32.730,156.119
C08942=1055.162,124.327,-82.275,171.493,32.732,156.119
C08943=1055.168,124.576,-82.295,171.495,32.735,156.119
C08944=1055.174,124.825,-82.315,171.497,32.737,156.120
C08945=1055.180,125.075,-82.335,171.498,32.739,156.120
C08946=1055.186,125.324,-82.356,171.500,32.742,156.121
C08947=1055.192,125.572,-82.376,171.502,32.744,156.121
C08948=1055.199,125.858,-82.400,171.504,32.747,156.121
C08949=1055.206,126.143,-82.423,171.506,32.750,156.122
C08950=1055.212,126.428,-82.447,171.508,32.752,156.122
C08951=1055.220,126.713,-82.470,171.510,32.755,156.123
C08952=1055.226,126.963,-82.490,171.512,32.758,156.123
C08953=1055.232,127.212,-82.510,171.514,32.760,156.123
C08954=1055.238,127.460,-82.530,171.515,32.762,156.124
C08955=1055.244,127.710,-82.552,171.516,32.765,156.124
C08956=1055.250,127.958,-82.572,171.518,32.767,156.125
C08957=1055.256,128.208,-82.592,171.520,32.769,156.125
C08958=1055.262,128.457,-82.613,171.522,32.771,156.125
C08959=1055.268,128.706,-82.634,171.523,32.774,156.126
C08960=1055.274,128.955,-82.654,171.525,32.776,156.126
C08961=1055.280,129.205,-82.675,171.527,32.778,156.127
C08962=1055.286,129.453,-82.695,171.529,32.781,156.127
C08963=1055.292,129.702,-82.716,171.531,32.784,156.127
C08964=1055.298,129.951,-82.736,171.532,32.786,156.128
C08965=1055.304,130.200,-82.756,171.534,32.788,156.128
C08966=1055.311,130.449,-82.778,171.536,32.790,156.129
C08967=1055.317,130.698,-82.798,171.538,32.793,156.129
C08968=1055.323,130.948,-82.818,171.540,32.795,156.129
C08969=1055.329,131.196,-82.840,171.541,32.797,156.130
C08970=1055.335,131.446,-82.860,171.543,32.800,156.130
C08971=1055.341,131.695,-82.880,171.545,32.802,156.131
C08972=1055.348,131.944,-82.901,171.547,32.804,156.131
C08973=1055.353,132.193,-82.922,171.549,32.807,156.131
C08974=1055.359,132.442,-82.942,171.550,32.810,156.132
C08975=1055.365,132.691,-82.964,171.552,32.812,156.132
C08976=1055.371,132.941,-82.984,171.554,32.814,156.132
C08977=1055.377,133.189,-83.005,171.556,32.817,156.133
C08978=1055.383,133.439,-83.026,171.558,32.819,156.133
C08979=1055.389,133.687,-83.047,171.559,32.822,156.134
C08980=1055.395,133.936,-83.067,171.561,32.824,156.134
C08981=1055.401,134.185,-83.089,171.563,32.826,156.135
C08982=1055.406,134.434,-83.110,171.565,32.829,156.135
C08983=1055.413,134.683,-83.131,171.567,32.832,156.135
C08984=1055.418,134.932,-83.151,171.568,32.833,156.136
C08985=1055.424,135.182,-83.173,171.570,32.836,156.136
C08986=1055.430,135.431,-83.193,171.572,32.839,156.137
C08987=1055.436,135.680,-83.214,171.574,32.841,156.137
C08988=1055.442,135.929,-83.235,171.576,32.843,156.137
C08989=1055.449,136.178,-83.256,171.577,32.846,156.138
C08990=1055.454,136.428,-83.277,171.579,32.848,156.138
C08991=1055.460,136.676,-83.298,171.581,32.851,156.139
C08992=1055.467,136.926,-83.318,171.583,32.853,156.139
C08993=1055.472,137.174,-83.340,171.584,32.856,156.139
C08994=1055.478,137.423,-83.361,171.586,32.858,156.140
C08995=1055.484,137.672,-83.381,171.587,32.860,156.140
C08996=1055.490,137.921,-83.403,171.589,32.863,156.141
C08997=1055.496,138.170,-83.423,171.591,32.865,156.141
C08998=1055.502,138.420,-83.445,171.593,32.868,156.141
C08999=1055.508,138.668,-83.466,171.595,32.870,156.142
C09000=1055.514,138.918,-83.487,171.597,32.872,156.142
C09001=1055.520,139.167,-83.508,171.598,32.875,156.143
C09002=1055.526,139.415,-83.530,171.600,32.877,156.143
C09003=1055.532,139.665,-83.550,171.602,32.880,156.143
C09004=1055.538,139.913,-83.571,171.604,32.882,156.144
C09005=1055.544,140.163,-83.593,171.606,32.885,156.144
C09006=1055.549,140.412,-83.613,171.608,32.887,156.145
C09007=1055.555,140.661,-83.635,171.609,32.890,156.145
C09008=1055.561,140.909,-83.656,171.611,32.892,156.146
C09009=1055.567,141.159,-83.678,171.613,32.894,156.146
C09010=1055.574,141.408,-83.698,171.615,32.897,156.146
C09011=1055.579,141.657,-83.720,171.617,32.899,156.147
C09012=1055.586,141.942,-83.745,171.619,32.902,156.147
C09013=1055.593,142.227,-83.768,171.621,32.905,156.148
C09014=1055.600,142.512,-83.793,171.623,32.908,156.148
C09015=1055.607,142.797,-83.817,171.625,32.911,156.149
C09016=1055.612,143.045,-83.839,171.627,32.913,156.149
C09017=1055.618,143.295,-83.860,171.629,32.916,156.149
C09018=1055.624,143.544,-83.881,171.631,32.918,156.150
C09019=1055.630,143.793,-83.903,171.633,32.921,156.150
C09020=1055.636,144.042,-83.924,171.634,32.923,156.151
C09021=1055.642,144.291,-83.945,171.636,32.926,156.151
C09022=1055.648,144.540,-83.967,171.638,32.928,156.151
C09023=1055.654,144.789,-83.989,171.640,32.930,156.152
C09024=1055.660,145.038,-84.009,171.642,32.933,156.152
C09025=1055.666,145.287,-84.030,171.644,32.936,156.153
C09026=1055.672,145.536,-84.052,171.646,32.938,156.153
C09027=1055.678,145.785,-84.073,171.648,32.940,156.154
C09028=1055.684,146.034,-84.095,171.649,32.943,156.154
C09029=1055.690,146.283,-84.117,171.651,32.945,156.154
C09030=1055.696,146.532,-84.138,171.653,32.948,156.155
C09031=1055.702,146.781,-84.159,171.655,32.950,156.155
C09032=1055.708,147.030,-84.181,171.657,32.952,156.156
C09033=1055.714,147.279,-84.202,171.659,32.955,156.156
C09034=1055.720,147.528,-84.224,171.661,32.958,156.156
C09035=1055.726,147.777,-84.246,171.663,32.960,156.157
C09036=1055.732,148.026,-84.267,171.664,32.963,156.157
C09037=1055.738,148.275,-84.289,171.666,32.965,156.158
C09038=1055.744,148.524,-84.310,171.668,32.967,156.158
C09039=1055.750,148.773,-84.332,171.670,32.970,156.158
C09040=1055.756,149.022,-84.353,171.672,32.972,156.159
C09041=1055.761,149.271,-84.375,171.674,32.975,156.159
C09042=1055.767,149.520,-84.397,171.676,32.978,156.160
C09043=1055.773,149.769,-84.418,171.678,32.980,156.160
C09044=1055.779,150.018,-84.440,171.679,32.983,156.161
C09045=1055.785,150.267,-84.461,171.681,32.985,156.161
C09046=1055.791,150.516,-84.483,171.683,32.988,156.162
C09047=1055.797,150.765,-84.504,171.685,32.990,156.162
C09048=1055.803,151.014,-84.527,171.687,32.992,156.162
C09049=1055.809,151.263,-84.549,171.689,32.995,156.163
C09050=1055.814,151.512,-84.570,171.691,32.997,156.163
C09051=1055.820,151.761,-84.592,171.693,33.000,156.164
C09052=1055.827,152.010,-84.613,171.695,33.003,156.164
C09053=1055.833,152.259,-84.635,171.697,33.005,156.164
C09054=1055.838,152.508,-84.657,171.698,33.008,156.165
C09055=1055.844,152.757,-84.679,171.700,33.010,156.165
C09056=1055.850,153.006,-84.701,171.702,33.013,156.166
C09057=1055.856,153.255,-84.723,171.704,33.015,156.166
C09058=1055.862,153.504,-84.744,171.705,33.017,156.167
C09059=1055.867,153.753,-84.766,171.707,33.020,156.167
C09060=1055.874,154.002,-84.788,171.709,33.023,156.167
C09061=1055.880,154.251,-84.810,171.711,33.025,156.168
C09062=1055.886,154.499,-84.831,171.713,33.028,156.168
